C07160=1017.237,129.736,-118.733,167.035,53.865,159.921
C07161=1017.243,129.986,-118.752,167.038,53.856,159.920
C07162=1017.248,130.235,-118.770,167.040,53.847,159.919
C07163=1017.252,130.484,-118.790,167.043,53.838,159.918
C07164=1017.258,130.733,-118.809,167.046,53.829,159.917
C07165=1017.262,130.983,-118.828,167.049,53.820,159.915
C07166=1017.267,131.232,-118.847,167.052,53.811,159.914
C07167=1017.272,131.480,-118.866,167.055,53.802,159.913
C07168=1017.276,131.731,-118.885,167.058,53.793,159.912
C07169=1017.282,131.980,-118.904,167.061,53.784,159.911
C07170=1017.286,132.229,-118.923,167.065,53.774,159.910
C07171=1017.291,132.478,-118.941,167.068,53.765,159.909
C07172=1017.296,132.728,-118.961,167.071,53.756,159.907
C07173=1017.301,132.976,-118.980,167.074,53.747,159.906
C07174=1017.306,133.225,-118.999,167.077,53.738,159.905
C07175=1017.310,133.476,-119.018,167.081,53.730,159.904
C07176=1017.315,133.724,-119.037,167.084,53.721,159.903
C07177=1017.320,133.973,-119.056,167.087,53.712,159.902
C07178=1017.325,134.222,-119.075,167.091,53.702,159.901
C07179=1017.330,134.472,-119.094,167.094,53.693,159.900
C07180=1017.335,134.721,-119.113,167.097,53.684,159.898
C07181=1017.340,134.970,-119.132,167.100,53.675,159.897
C07182=1017.345,135.220,-119.152,167.103,53.666,159.896
C07183=1017.350,135.468,-119.171,167.106,53.657,159.895
C07184=1017.354,135.718,-119.189,167.110,53.648,159.894
C07185=1017.360,135.967,-119.209,167.113,53.639,159.893
C07186=1017.364,136.216,-119.228,167.116,53.630,159.892
C07187=1017.369,136.465,-119.247,167.119,53.621,159.890
C07188=1017.375,136.715,-119.266,167.122,53.612,159.889
C07189=1017.379,136.964,-119.286,167.125,53.603,159.888
C07190=1017.385,137.213,-119.305,167.128,53.594,159.887
C07191=1017.389,137.463,-119.324,167.132,53.585,159.886
C07192=1017.394,137.712,-119.343,167.135,53.576,159.885
C07193=1017.399,137.961,-119.363,167.138,53.567,159.884
C07194=1017.403,138.210,-119.382,167.141,53.558,159.882
C07195=1017.408,138.459,-119.401,167.144,53.549,159.881
C07196=1017.414,138.741,-119.423,167.148,53.538,159.880
C07197=1017.419,139.022,-119.445,167.151,53.528,159.879
C07198=1017.424,139.304,-119.467,167.155,53.518,159.877
C07199=1017.430,139.585,-119.489,167.159,53.508,159.876
C07200=1017.434,139.834,-119.508,167.162,53.499,159.875
C07201=1017.440,140.084,-119.528,167.166,53.490,159.874
C07202=1017.444,140.333,-119.547,167.169,53.481,159.873
C07203=1017.449,140.583,-119.567,167.172,53.472,159.872
C07204=1017.454,140.831,-119.586,167.175,53.464,159.871
C07205=1017.459,141.080,-119.606,167.179,53.455,159.870
C07206=1017.464,141.329,-119.626,167.182,53.446,159.868
C07207=1017.469,141.578,-119.645,167.186,53.436,159.867
C07208=1017.474,141.828,-119.665,167.189,53.427,159.866
C07209=1017.478,142.077,-119.684,167.192,53.418,159.865
C07210=1017.484,142.326,-119.703,167.195,53.409,159.864
C07211=1017.488,142.575,-119.723,167.198,53.400,159.863
C07212=1017.493,142.825,-119.743,167.201,53.391,159.862
C07213=1017.498,143.074,-119.762,167.205,53.382,159.861
C07214=1017.503,143.323,-119.781,167.208,53.373,159.859
C07215=1017.508,143.572,-119.802,167.211,53.364,159.858
C07216=1017.512,143.821,-119.821,167.214,53.355,159.857
C07217=1017.518,144.071,-119.840,167.217,53.346,159.856
C07218=1017.522,144.320,-119.860,167.222,53.337,159.855
C07219=1017.527,144.569,-119.880,167.225,53.329,159.854
C07220=1017.532,144.818,-119.898,167.228,53.320,159.853
C07221=1017.538,145.067,-119.919,167.231,53.311,159.852
C07222=1017.542,145.316,-119.939,167.234,53.302,159.850
C07223=1017.548,145.566,-119.958,167.238,53.293,159.849
C07224=1017.552,145.815,-119.977,167.242,53.284,159.848
C07225=1017.557,146.064,-119.998,167.245,53.275,159.847
C07226=1017.562,146.313,-120.017,167.248,53.266,159.846
C07227=1017.567,146.563,-120.037,167.251,53.257,159.845
C07228=1017.571,146.812,-120.057,167.255,53.247,159.844
C07229=1017.576,147.061,-120.077,167.259,53.239,159.843
C07230=1017.581,147.310,-120.097,167.262,53.230,159.842
C07231=1017.586,147.559,-120.116,167.265,53.221,159.841
C07232=1017.592,147.808,-120.136,167.268,53.212,159.839
C07233=1017.596,148.057,-120.156,167.271,53.203,159.838
C07234=1017.601,148.307,-120.176,167.275,53.194,159.837
C07235=1017.605,148.556,-120.196,167.278,53.185,159.836
C07236=1017.610,148.805,-120.216,167.282,53.177,159.835
C07237=1017.615,149.054,-120.236,167.285,53.168,159.834
C07238=1017.620,149.304,-120.256,167.288,53.159,159.833
C07239=1017.625,149.552,-120.276,167.292,53.150,159.832
C07240=1017.630,149.802,-120.296,167.295,53.141,159.831
C07241=1017.635,150.051,-120.316,167.298,53.132,159.829
C07242=1017.639,150.300,-120.336,167.302,53.123,159.828
C07243=1017.644,150.549,-120.356,167.305,53.115,159.827
C07244=1017.649,150.798,-120.376,167.309,53.105,159.826
C07245=1017.654,151.048,-120.396,167.312,53.097,159.825
C07246=1017.658,151.296,-120.416,167.316,53.088,159.824
C07247=1017.663,151.546,-120.436,167.319,53.079,159.823
C07248=1017.669,151.795,-120.456,167.323,53.069,159.822
C07249=1017.673,152.044,-120.476,167.326,53.061,159.821
C07250=1017.678,152.293,-120.496,167.330,53.052,159.820
C07251=1017.684,152.542,-120.516,167.333,53.043,159.819
C07252=1017.689,152.791,-120.536,167.336,53.035,159.818
C07253=1017.693,153.041,-120.557,167.340,53.025,159.816
C07254=1017.697,153.290,-120.576,167.343,53.016,159.815
C07255=1017.703,153.539,-120.597,167.346,53.007,159.814
C07256=1017.708,153.788,-120.617,167.350,52.999,159.813
C07257=1017.712,154.037,-120.637,167.354,52.990,159.812
C07258=1017.718,154.286,-120.657,167.357,52.981,159.811
C07259=1017.723,154.536,-120.677,167.360,52.972,159.810
C07260=1017.728,154.817,-120.701,167.364,52.962,159.809
C07261=1017.733,155.099,-120.723,167.368,52.952,159.807
C07262=1017.739,155.380,-120.746,167.372,52.942,159.806
C07263=1017.744,155.662,-120.769,167.376,52.932,159.805
C07264=1017.749,155.910,-120.789,167.380,52.924,159.804
C07265=1017.754,156.159,-120.810,167.383,52.915,159.803
C07266=1017.759,156.408,-120.830,167.386,52.906,159.802
C07267=1017.764,156.657,-120.850,167.391,52.897,159.801
C07268=1017.769,156.906,-120.870,167.394,52.888,159.800
C07269=1017.774,157.156,-120.892,167.397,52.880,159.799
C07270=1017.778,157.405,-120.911,167.401,52.871,159.798
C07271=1017.783,157.654,-120.932,167.405,52.862,159.797
C07272=1017.788,157.903,-120.952,167.408,52.853,159.795
C07273=1017.794,158.152,-120.973,167.411,52.844,159.794
C07274=1017.798,158.401,-120.992,167.415,52.835,159.793
C07275=1017.803,158.650,-121.013,167.419,52.826,159.792
C07276=1017.808,158.900,-121.034,167.422,52.818,159.791
C07277=1017.812,159.149,-121.055,167.425,52.809,159.790
C07278=1017.817,159.398,-121.075,167.429,52.801,159.789
C07279=1017.821,159.647,-121.096,167.432,52.792,159.788
C07280=1017.827,159.896,-121.117,167.437,52.783,159.787
C07281=1017.831,160.145,-121.138,167.440,52.774,159.786
C07282=1017.835,160.394,-121.159,167.444,52.766,159.785
C07283=1017.841,160.643,-121.180,167.447,52.757,159.784
C07284=1017.845,160.892,-121.201,167.450,52.748,159.783
C07285=1017.850,161.141,-121.221,167.454,52.740,159.782
C07286=1017.854,161.390,-121.243,167.458,52.731,159.781
C07287=1017.859,161.640,-121.264,167.462,52.723,159.780
C07288=1017.864,161.889,-121.284,167.465,52.714,159.779
C07289=1017.868,162.137,-121.305,167.468,52.705,159.778
C07290=1017.873,162.387,-121.326,167.472,52.697,159.777
C07291=1017.878,162.636,-121.347,167.475,52.688,159.776
C07292=1017.882,162.885,-121.368,167.480,52.680,159.775
C07293=1017.887,163.133,-121.389,167.483,52.671,159.774
C07294=1017.892,163.383,-121.410,167.486,52.662,159.772
C07295=1017.897,163.632,-121.431,167.490,52.654,159.772
C07296=1017.902,163.881,-121.452,167.494,52.645,159.771
C07297=1017.906,164.131,-121.473,167.498,52.637,159.770
C07298=1017.911,164.379,-121.493,167.501,52.628,159.768
C07299=1017.916,164.628,-121.515,167.504,52.619,159.767
C07300=1017.921,164.877,-121.535,167.508,52.611,159.766
C07301=1017.925,165.127,-121.557,167.512,52.602,159.765
C07302=1017.930,165.376,-121.578,167.516,52.593,159.764
C07303=1017.935,165.625,-121.598,167.519,52.585,159.763
C07304=1017.939,165.873,-121.620,167.523,52.575,159.762
C07305=1017.945,166.122,-121.640,167.527,52.567,159.761
C07306=1017.949,166.372,-121.662,167.530,52.558,159.760
C07307=1017.954,166.621,-121.683,167.534,52.550,159.759
C07308=1017.959,166.870,-121.704,167.538,52.541,159.758
C07309=1017.964,167.119,-121.725,167.542,52.532,159.757
C07310=1017.969,167.368,-121.746,167.545,52.524,159.756
C07311=1017.974,167.618,-121.767,167.548,52.515,159.755
C07312=1017.978,167.866,-121.788,167.553,52.506,159.754
C07313=1017.983,168.115,-121.809,167.556,52.498,159.753
C07314=1017.988,168.364,-121.830,167.560,52.489,159.752
C07315=1017.993,168.613,-121.851,167.564,52.480,159.751
C07316=1017.998,168.862,-121.872,167.568,52.472,159.750
C07317=1018.002,169.112,-121.894,167.571,52.463,159.749
C07318=1018.008,169.360,-121.915,167.575,52.454,159.748
C07319=1018.012,169.610,-121.936,167.579,52.446,159.747
C07320=1018.017,169.859,-121.957,167.582,52.437,159.746
C07321=1018.022,170.108,-121.978,167.587,52.429,159.745
C07322=1018.027,170.357,-122.000,167.590,52.420,159.744
C07323=1018.032,170.606,-122.020,167.594,52.411,159.743
C07324=1018.038,170.887,-122.044,167.598,52.401,159.742
C07325=1018.043,171.168,-122.068,167.603,52.392,159.741
C07326=1018.048,171.449,-122.092,167.607,52.382,159.739
C07327=1018.054,171.731,-122.116,167.611,52.372,159.738
C07328=1018.058,171.980,-122.137,167.615,52.364,159.737
C07329=1018.064,172.228,-122.158,167.618,52.355,159.736
C07330=1018.069,172.478,-122.180,167.623,52.346,159.735
C07331=1018.074,172.727,-122.201,167.627,52.338,159.734
C07332=1018.079,172.976,-122.222,167.630,52.329,159.733
C07333=1018.084,173.225,-122.244,167.634,52.320,159.732
C07334=1018.089,173.474,-122.265,167.638,52.312,159.731
C07335=1018.094,173.723,-122.287,167.642,52.302,159.730
C07336=1018.098,173.972,-122.308,167.645,52.294,159.729
C07337=1018.104,174.221,-122.329,167.649,52.286,159.728
C07338=1018.108,174.470,-122.350,167.654,52.276,159.727
C07339=1018.114,174.719,-122.371,167.657,52.268,159.726
C07340=1018.118,174.968,-122.393,167.662,52.259,159.725
C07341=1018.123,175.217,-122.414,167.665,52.250,159.724
C07342=1018.129,175.466,-122.435,167.669,52.241,159.723
C07343=1018.133,175.715,-122.457,167.673,52.233,159.722
C07344=1018.138,175.964,-122.478,167.676,52.225,159.721
C07345=1018.143,176.213,-122.499,167.681,52.215,159.720
C07346=1018.148,176.462,-122.521,167.684,52.207,159.719
C07347=1018.154,176.711,-122.542,167.689,52.198,159.718
C07348=1018.159,176.960,-122.564,167.692,52.190,159.717
C07349=1018.163,177.210,-122.585,167.697,52.181,159.716
C07350=1018.169,177.458,-122.606,167.700,52.172,159.715
C07351=1018.174,177.707,-122.628,167.705,52.164,159.714
C07352=1018.178,177.956,-122.649,167.708,52.155,159.713
C07353=1018.184,178.205,-122.671,167.713,52.146,159.712
C07354=1018.189,178.454,-122.693,167.716,52.138,159.711
C07355=1018.194,178.704,-122.714,167.721,52.129,159.710
C07356=1018.199,178.952,-122.735,167.724,52.120,159.709
C07357=1018.204,179.201,-122.757,167.729,52.112,159.708
C07358=1018.210,179.450,-122.778,167.732,52.103,159.707
C07359=1018.214,179.699,-122.800,167.737,52.094,159.706
C07360=1018.220,179.949,-122.822,167.740,52.086,159.705
C07361=1018.225,180.198,-122.842,167.745,52.077,159.704
C07362=1018.230,180.447,-122.864,167.748,52.068,159.703
C07363=1018.235,180.695,-122.886,167.753,52.060,159.702
C07364=1018.240,180.944,-122.907,167.756,52.051,159.701
C07365=1018.245,181.194,-122.929,167.761,52.042,159.700
C07366=1018.250,181.443,-122.951,167.764,52.034,159.699
C07367=1018.256,181.691,-122.972,167.769,52.025,159.698
C07368=1018.261,181.940,-122.994,167.772,52.016,159.697
C07369=1018.266,182.190,-123.016,167.777,52.008,159.696
C07370=1018.270,182.439,-123.039,167.781,52.000,159.695
C07371=1018.275,182.688,-123.060,167.785,51.991,159.694
C07372=1018.280,182.937,-123.082,167.789,51.983,159.693
C07373=1018.284,183.186,-123.105,167.793,51.975,159.692
C07374=1018.289,183.435,-123.127,167.797,51.965,159.691
C07375=1018.294,183.684,-123.149,167.801,51.957,159.690
C07376=1018.299,183.933,-123.171,167.805,51.949,159.689
C07377=1018.303,184.182,-123.193,167.809,51.941,159.688
C07378=1018.309,184.431,-123.216,167.813,51.932,159.687
C07379=1018.314,184.680,-123.238,167.818,51.924,159.686
C07380=1018.318,184.928,-123.260,167.821,51.916,159.685
C07381=1018.322,185.178,-123.282,167.825,51.907,159.684
C07382=1018.328,185.427,-123.305,167.830,51.899,159.684
C07383=1018.333,185.675,-123.327,167.833,51.891,159.683
C07384=1018.337,185.924,-123.350,167.838,51.882,159.682
C07385=1018.342,186.173,-123.371,167.842,51.874,159.681
C07386=1018.347,186.423,-123.394,167.846,51.865,159.680
C07387=1018.351,186.672,-123.416,167.850,51.857,159.679
C07388=1018.357,186.952,-123.441,167.854,51.848,159.678
C07389=1018.363,187.233,-123.467,167.860,51.838,159.677
C07390=1018.368,187.514,-123.492,167.864,51.829,159.676
C07391=1018.374,187.794,-123.517,167.869,51.819,159.675
C07392=1018.379,188.044,-123.539,167.872,51.811,159.674
C07393=1018.384,188.292,-123.561,167.877,51.802,159.673
C07394=1018.388,188.541,-123.584,167.881,51.794,159.672
C07395=1018.394,188.790,-123.607,167.886,51.785,159.671
C07396=1018.398,189.039,-123.629,167.889,51.777,159.670
C07397=1018.403,189.288,-123.652,167.894,51.769,159.669
C07398=1018.408,189.537,-123.674,167.898,51.761,159.668
C07399=1018.413,189.786,-123.696,167.903,51.752,159.667
C07400=1018.419,190.035,-123.719,167.906,51.744,159.666
C07401=1018.423,190.284,-123.741,167.911,51.736,159.665
C07402=1018.428,190.533,-123.763,167.915,51.727,159.664
C07403=1018.433,190.782,-123.786,167.919,51.719,159.663
C07404=1018.438,191.031,-123.808,167.923,51.711,159.662
C07405=1018.443,191.280,-123.831,167.928,51.702,159.661
C07406=1018.448,191.529,-123.853,167.932,51.694,159.661
C07407=1018.453,191.777,-123.876,167.936,51.685,159.660
C07408=1018.458,192.027,-123.899,167.940,51.677,159.659
C07409=1018.463,192.275,-123.921,167.945,51.668,159.658
C07410=1018.468,192.525,-123.944,167.949,51.660,159.657
C07411=1018.473,192.773,-123.966,167.953,51.651,159.656
C07412=1018.478,193.022,-123.989,167.958,51.643,159.655
C07413=1018.483,193.271,-124.011,167.962,51.635,159.654
C07414=1018.488,193.520,-124.034,167.967,51.627,159.653
C07415=1018.493,193.769,-124.056,167.970,51.618,159.652
C07416=1018.498,194.017,-124.079,167.975,51.610,159.651
C07417=1018.503,194.267,-124.102,167.980,51.602,159.651
C07418=1018.508,194.515,-124.124,167.983,51.593,159.649
C07419=1018.514,194.764,-124.147,167.988,51.585,159.649
C07420=1018.518,195.014,-124.170,167.992,51.577,159.648
C07421=1018.523,195.262,-124.192,167.996,51.568,159.647
C07422=1018.529,195.512,-124.215,168.001,51.559,159.646
C07423=1018.533,195.760,-124.238,168.005,51.551,159.645
C07424=1018.539,196.009,-124.261,168.010,51.543,159.644
C07425=1018.544,196.258,-124.283,168.013,51.535,159.643
C07426=1018.549,196.507,-124.306,168.018,51.526,159.642
C07427=1018.554,196.756,-124.328,168.023,51.518,159.641
C07428=1018.559,197.005,-124.351,168.027,51.509,159.640
C07429=1018.564,197.253,-124.374,168.032,51.501,159.639
C07430=1018.569,197.503,-124.396,168.036,51.493,159.639
C07431=1018.575,197.752,-124.419,168.040,51.485,159.638
C07432=1018.580,198.000,-124.442,168.045,51.476,159.637
C07433=1018.585,198.249,-124.466,168.050,51.468,159.636
C07434=1018.590,198.498,-124.487,168.054,51.460,159.635
C07435=1018.596,198.747,-124.510,168.058,51.451,159.634
C07436=1018.601,198.996,-124.534,168.063,51.442,159.633
C07437=1018.605,199.245,-124.556,168.068,51.434,159.632
C07438=1018.610,199.494,-124.579,168.072,51.426,159.631
C07439=1018.616,199.743,-124.602,168.077,51.418,159.630
C07440=1018.621,199.992,-124.625,168.081,51.410,159.630
C07441=1018.625,200.241,-124.649,168.085,51.402,159.629
C07442=1018.631,200.490,-124.672,168.090,51.393,159.628
C07443=1018.636,200.738,-124.695,168.094,51.385,159.627
C07444=1018.641,200.987,-124.719,168.099,51.377,159.626
C07445=1018.645,201.236,-124.742,168.103,51.369,159.625
C07446=1018.651,201.485,-124.765,168.108,51.361,159.624
C07447=1018.656,201.734,-124.788,168.112,51.352,159.623
C07448=1018.660,201.983,-124.811,168.116,51.344,159.622
C07449=1018.666,202.231,-124.834,168.121,51.336,159.622
C07450=1018.671,202.481,-124.858,168.126,51.328,159.621
C07451=1018.675,202.729,-124.881,168.130,51.320,159.620
C07452=1018.702,203.979,-125.000,168.600,51.411,159.725
C07453=1018.707,204.207,-125.023,168.603,51.404,159.724
C07454=1018.713,204.434,-125.045,168.607,51.398,159.723
C07455=1018.718,204.661,-125.068,168.610,51.391,159.723
C07456=1018.724,204.888,-125.090,168.614,51.385,159.722
C07457=1018.730,205.116,-125.113,168.617,51.378,159.721
C07458=1018.735,205.343,-125.137,168.620,51.372,159.720
C07459=1018.740,205.570,-125.159,168.624,51.365,159.720
C07460=1018.747,205.819,-125.184,168.628,51.358,159.719
C07461=1018.753,206.068,-125.209,168.631,51.351,159.718
C07462=1018.758,206.316,-125.234,168.635,51.343,159.717
C07463=1018.764,206.565,-125.259,168.640,51.336,159.716
C07464=1018.771,206.813,-125.284,168.643,51.329,159.715
C07465=1018.777,207.062,-125.310,168.647,51.322,159.715
C07466=1018.782,207.311,-125.334,168.650,51.315,159.714
C07467=1018.788,207.559,-125.359,168.655,51.308,159.713
C07468=1018.794,207.808,-125.385,168.658,51.301,159.712
C07469=1018.801,208.057,-125.410,168.662,51.294,159.711
C07470=1018.806,208.305,-125.435,168.666,51.287,159.711
C07471=1018.812,208.554,-125.460,168.670,51.280,159.710
C07472=1018.818,208.803,-125.485,168.674,51.273,159.709
C07473=1018.824,209.052,-125.511,168.677,51.266,159.708
C07474=1018.830,209.300,-125.536,168.682,51.260,159.707
C07475=1018.836,209.548,-125.561,168.685,51.253,159.707
C07476=1018.842,209.797,-125.586,168.689,51.246,159.706
C07477=1018.848,210.046,-125.612,168.692,51.239,159.705
C07478=1018.854,210.294,-125.637,168.697,51.232,159.704
C07479=1018.860,210.543,-125.663,168.700,51.225,159.703
C07480=1018.866,210.792,-125.688,168.705,51.218,159.703
C07481=1018.872,211.040,-125.713,168.708,51.212,159.702
C07482=1018.878,211.289,-125.739,168.712,51.204,159.701
C07483=1018.883,211.538,-125.765,168.715,51.198,159.700
C07484=1018.889,211.786,-125.790,168.720,51.191,159.700
C07485=1018.896,212.035,-125.815,168.723,51.184,159.699
C07486=1018.901,212.284,-125.841,168.728,51.177,159.698
C07487=1018.907,212.533,-125.867,168.731,51.170,159.697
C07488=1018.913,212.781,-125.892,168.735,51.164,159.696
C07489=1018.919,213.029,-125.917,168.739,51.157,159.696
C07490=1018.925,213.278,-125.943,168.742,51.150,159.695
C07491=1018.931,213.527,-125.968,168.747,51.144,159.694
C07492=1018.937,213.775,-125.994,168.750,51.137,159.693
C07493=1018.942,214.024,-126.019,168.754,51.130,159.693
C07494=1018.949,214.273,-126.045,168.758,51.124,159.692
C07495=1018.955,214.521,-126.071,168.762,51.117,159.691
C07496=1018.961,214.770,-126.096,168.765,51.110,159.690
C07497=1018.967,215.019,-126.122,168.770,51.103,159.690
C07498=1018.973,215.268,-126.147,168.773,51.096,159.689
C07499=1018.979,215.516,-126.173,168.777,51.090,159.688
C07500=1018.984,215.764,-126.198,168.781,51.083,159.687
C07501=1018.990,216.013,-126.224,168.785,51.076,159.687
C07502=1018.997,216.261,-126.250,168.789,51.070,159.686
C07503=1019.003,216.510,-126.275,168.793,51.063,159.685
C07504=1019.009,216.759,-126.301,168.797,51.057,159.685
C07505=1019.015,217.007,-126.326,168.801,51.050,159.684
C07506=1019.021,217.256,-126.352,168.805,51.043,159.683
C07507=1019.027,217.505,-126.378,168.809,51.037,159.682
C07508=1019.033,217.753,-126.404,168.812,51.031,159.682
C07509=1019.039,218.002,-126.429,168.816,51.023,159.681
C07510=1019.046,218.250,-126.455,168.820,51.017,159.680
C07511=1019.051,218.499,-126.481,168.824,51.010,159.679
C07512=1019.057,218.726,-126.505,168.827,51.004,159.679
C07513=1019.062,218.955,-126.528,168.831,50.999,159.678
C07514=1019.068,219.183,-126.552,168.835,50.993,159.677
C07515=1019.073,219.411,-126.577,168.839,50.987,159.677
C07516=1019.078,219.639,-126.600,168.842,50.981,159.676
C07517=1019.084,219.867,-126.624,168.846,50.975,159.676
C07518=1019.089,220.095,-126.648,168.849,50.969,159.675
C07519=1019.095,220.322,-126.672,168.853,50.963,159.674
C07520=1019.100,220.571,-126.698,168.856,50.957,159.674
C07521=1019.107,220.819,-126.724,168.861,50.950,159.673
C07522=1019.112,221.068,-126.750,168.864,50.944,159.672
C07523=1019.118,221.317,-126.777,168.868,50.938,159.671
C07524=1019.124,221.565,-126.802,168.873,50.931,159.671
C07525=1019.131,221.814,-126.829,168.876,50.925,159.670
C07526=1019.137,222.063,-126.854,168.880,50.919,159.669
C07527=1019.143,222.311,-126.881,168.884,50.912,159.669
C07528=1019.148,222.560,-126.907,168.888,50.906,159.668
C07529=1019.155,222.808,-126.933,168.892,50.900,159.667
C07530=1019.160,223.057,-126.959,168.897,50.894,159.667
C07531=1019.167,223.305,-126.985,168.900,50.887,159.666
C07532=1019.172,223.554,-127.012,168.904,50.881,159.665
C07533=1019.178,223.803,-127.038,168.908,50.874,159.665
C07534=1019.185,224.052,-127.064,168.912,50.868,159.664
C07535=1019.190,224.300,-127.090,168.916,50.862,159.663
C07536=1019.197,224.549,-127.116,168.920,50.856,159.663
C07537=1019.203,224.797,-127.143,168.924,50.850,159.662
C07538=1019.208,225.046,-127.168,168.928,50.843,159.662
C07539=1019.215,225.294,-127.195,168.932,50.836,159.661
C07540=1019.220,225.542,-127.221,168.936,50.830,159.660
C07541=1019.227,225.792,-127.247,168.940,50.824,159.659
C07542=1019.233,226.040,-127.274,168.944,50.818,159.659
C07543=1019.239,226.288,-127.300,168.948,50.812,159.658
C07544=1019.245,226.536,-127.326,168.952,50.806,159.658
C07545=1019.251,226.785,-127.352,168.955,50.800,159.657
C07546=1019.257,227.034,-127.379,168.960,50.793,159.656
C07547=1019.263,227.283,-127.406,168.964,50.787,159.656
C07548=1019.269,227.531,-127.432,168.967,50.781,159.655
C07549=1019.275,227.779,-127.459,168.972,50.776,159.655
C07550=1019.281,228.028,-127.485,168.976,50.769,159.654
C07551=1019.287,228.276,-127.512,168.980,50.763,159.653
C07552=1019.293,228.526,-127.538,168.984,50.757,159.653
C07553=1019.299,228.774,-127.565,168.987,50.751,159.652
C07554=1019.305,229.022,-127.591,168.992,50.745,159.651
C07555=1019.311,229.270,-127.617,168.996,50.738,159.651
C07556=1019.317,229.519,-127.645,169.000,50.733,159.650
C07557=1019.323,229.768,-127.671,169.004,50.727,159.650
C07558=1019.329,230.016,-127.698,169.007,50.721,159.649
C07559=1019.335,230.265,-127.724,169.012,50.715,159.648
C07560=1019.341,230.514,-127.751,169.016,50.709,159.648
C07561=1019.347,230.762,-127.778,169.020,50.703,159.647
C07562=1019.353,231.010,-127.805,169.024,50.697,159.647
C07563=1019.358,231.259,-127.831,169.028,50.692,159.646
C07564=1019.365,231.508,-127.858,169.033,50.685,159.646
C07565=1019.371,231.755,-127.886,169.036,50.679,159.645
C07566=1019.377,232.004,-127.912,169.040,50.674,159.644
C07567=1019.383,232.253,-127.939,169.044,50.668,159.644
C07568=1019.389,232.501,-127.966,169.048,50.662,159.643
C07569=1019.394,232.750,-127.993,169.053,50.656,159.643
C07570=1019.400,232.998,-128.019,169.057,50.650,159.642
C07571=1019.407,233.247,-128.046,169.060,50.644,159.641
C07572=1019.412,233.470,-128.071,169.064,50.639,159.641
C07573=1019.418,233.695,-128.095,169.068,50.633,159.640
C07574=1019.423,233.918,-128.119,169.072,50.628,159.640
C07575=1019.429,234.143,-128.143,169.075,50.623,159.639
C07576=1019.434,234.366,-128.167,169.079,50.618,159.639
C07577=1019.440,234.590,-128.192,169.082,50.613,159.638
C07578=1019.445,234.814,-128.216,169.086,50.607,159.638
C07579=1019.450,235.038,-128.241,169.089,50.602,159.637
C07580=1019.456,235.286,-128.268,169.094,50.596,159.637
C07581=1019.462,235.534,-128.294,169.098,50.590,159.636
C07582=1019.468,235.783,-128.322,169.102,50.585,159.636
C07583=1019.474,236.031,-128.349,169.106,50.579,159.635
C07584=1019.481,236.280,-128.376,169.110,50.574,159.635
C07585=1019.487,236.528,-128.403,169.114,50.568,159.634
C07586=1019.492,236.776,-128.430,169.119,50.562,159.634
C07587=1019.499,237.025,-128.457,169.123,50.556,159.633
C07588=1019.505,237.273,-128.484,169.127,50.551,159.632
C07589=1019.511,237.522,-128.511,169.131,50.545,159.632
C07590=1019.517,237.771,-128.538,169.135,50.539,159.631
C07591=1019.524,238.019,-128.566,169.139,50.534,159.631
C07592=1019.529,238.267,-128.592,169.144,50.527,159.630
C07593=1019.535,238.516,-128.619,169.148,50.522,159.630
C07594=1019.541,238.765,-128.647,169.152,50.517,159.629
C07595=1019.547,239.013,-128.674,169.156,50.511,159.629
C07596=1019.554,239.261,-128.702,169.160,50.505,159.628
C07597=1019.559,239.510,-128.728,169.164,50.500,159.628
C07598=1019.565,239.758,-128.756,169.168,50.495,159.627
C07599=1019.571,240.007,-128.783,169.172,50.489,159.627
C07600=1019.578,240.255,-128.811,169.176,50.483,159.626
C07601=1019.583,240.503,-128.839,169.180,50.478,159.626
C07602=1019.590,240.752,-128.866,169.185,50.472,159.625
C07603=1019.596,241.000,-128.893,169.189,50.467,159.625
C07604=1019.602,241.249,-128.922,169.194,50.461,159.624
C07605=1019.607,241.497,-128.948,169.197,50.455,159.624
C07606=1019.614,241.746,-128.976,169.201,50.450,159.623
C07607=1019.619,241.994,-129.004,169.206,50.445,159.623
C07608=1019.626,242.243,-129.031,169.210,50.439,159.622
C07609=1019.632,242.491,-129.058,169.214,50.434,159.622
C07610=1019.638,242.739,-129.087,169.218,50.429,159.621
C07611=1019.644,242.988,-129.113,169.222,50.423,159.621
C07612=1019.650,243.236,-129.141,169.226,50.418,159.620
C07613=1019.656,243.484,-129.169,169.230,50.413,159.620
C07614=1019.661,243.733,-129.197,169.235,50.407,159.620
C07615=1019.668,243.981,-129.225,169.239,50.402,159.619
C07616=1019.673,244.230,-129.252,169.243,50.397,159.619
C07617=1019.679,244.478,-129.280,169.247,50.391,159.618
C07618=1019.685,244.726,-129.308,169.251,50.386,159.618
C07619=1019.691,244.975,-129.336,169.255,50.381,159.617
C07620=1019.697,245.223,-129.364,169.259,50.375,159.617
C07621=1019.703,245.472,-129.392,169.264,50.370,159.616
C07622=1019.709,245.720,-129.420,169.268,50.365,159.616
C07623=1019.715,245.968,-129.448,169.272,50.360,159.616
C07624=1019.721,246.217,-129.476,169.276,50.355,159.615
C07625=1019.726,246.465,-129.504,169.280,50.349,159.615
C07626=1019.733,246.713,-129.532,169.285,50.344,159.614
C07627=1019.739,246.962,-129.560,169.289,50.339,159.614
C07628=1019.744,247.210,-129.588,169.293,50.334,159.613
C07629=1019.751,247.459,-129.616,169.297,50.329,159.613
C07630=1019.756,247.707,-129.644,169.302,50.323,159.612
C07631=1019.762,247.956,-129.672,169.307,50.318,159.612
C07632=1019.768,248.176,-129.696,169.310,50.313,159.612
C07633=1019.773,248.397,-129.722,169.314,50.309,159.611
C07634=1019.779,248.617,-129.746,169.318,50.304,159.611
C07635=1019.784,248.838,-129.771,169.321,50.299,159.610
C07636=1019.790,249.059,-129.796,169.325,50.295,159.610
C07637=1019.794,249.279,-129.821,169.330,50.290,159.610
C07638=1019.801,249.500,-129.846,169.333,50.286,159.610
C07639=1019.805,249.721,-129.871,169.337,50.282,159.609
C07640=1019.812,249.968,-129.899,169.341,50.276,159.609
C07641=1019.818,250.216,-129.927,169.345,50.271,159.608
C07642=1019.824,250.465,-129.956,169.349,50.266,159.608
C07643=1019.830,250.714,-129.983,169.354,50.261,159.607
C07644=1019.836,250.962,-130.012,169.358,50.256,159.607
C07645=1019.842,251.210,-130.040,169.362,50.251,159.607
C07646=1019.849,251.458,-130.068,169.366,50.246,159.606
C07647=1019.854,251.707,-130.096,169.371,50.240,159.606
C07648=1019.860,251.956,-130.125,169.375,50.236,159.606
C07649=1019.867,252.204,-130.152,169.379,50.230,159.605
C07650=1019.873,252.452,-130.181,169.384,50.226,159.605
C07651=1019.879,252.700,-130.210,169.388,50.220,159.604
C07652=1019.885,252.949,-130.237,169.392,50.215,159.604
C07653=1019.891,253.198,-130.266,169.397,50.210,159.604
C07654=1019.897,253.445,-130.294,169.401,50.205,159.603
C07655=1019.904,253.694,-130.322,169.405,50.200,159.603
C07656=1019.910,253.942,-130.350,169.410,50.195,159.602
C07657=1019.916,254.190,-130.379,169.414,50.191,159.602
C07658=1019.923,254.439,-130.407,169.418,50.185,159.602
C07659=1019.928,254.688,-130.435,169.423,50.181,159.601
C07660=1019.934,254.935,-130.464,169.427,50.175,159.601
C07661=1019.941,255.183,-130.492,169.431,50.171,159.601
C07662=1019.947,255.432,-130.520,169.436,50.165,159.600
C07663=1019.953,255.680,-130.549,169.440,50.161,159.600
C07664=1019.960,255.929,-130.577,169.444,50.155,159.599
C07665=1019.966,256.177,-130.606,169.449,50.151,159.599
C07666=1019.972,256.426,-130.634,169.453,50.145,159.599
C07667=1019.979,256.673,-130.663,169.458,50.141,159.598
C07668=1019.985,256.922,-130.691,169.462,50.136,159.598
C07669=1019.990,257.170,-130.719,169.467,50.131,159.598
C07670=1019.997,257.418,-130.747,169.472,50.126,159.597
C07671=1020.003,257.667,-130.776,169.476,50.121,159.597
C07672=1020.009,257.915,-130.805,169.481,50.116,159.597
C07673=1020.016,258.163,-130.833,169.485,50.111,159.596
C07674=1020.022,258.412,-130.862,169.489,50.106,159.596
C07675=1020.029,258.660,-130.891,169.494,50.101,159.596
C07676=1020.035,258.908,-130.918,169.498,50.097,159.595
C07677=1020.041,259.156,-130.947,169.503,50.091,159.595
C07678=1020.047,259.405,-130.976,169.507,50.087,159.595
C07679=1020.054,259.653,-131.004,169.512,50.082,159.594
C07680=1020.060,259.902,-131.032,169.516,50.077,159.594
C07681=1020.067,260.150,-131.062,169.520,50.072,159.594
C07682=1020.073,260.398,-131.091,169.525,50.068,159.593
C07683=1020.079,260.646,-131.120,169.529,50.063,159.593
C07684=1020.085,260.894,-131.149,169.533,50.059,159.593
C07685=1020.091,261.143,-131.177,169.538,50.054,159.592
C07686=1020.097,261.391,-131.206,169.542,50.049,159.592
C07687=1020.104,261.639,-131.235,169.547,50.045,159.592
C07688=1020.110,261.887,-131.264,169.551,50.040,159.592
C07689=1020.116,262.135,-131.293,169.556,50.036,159.591
C07690=1020.122,262.384,-131.323,169.560,50.031,159.591
C07691=1020.128,262.632,-131.352,169.565,50.026,159.591
C07692=1020.134,262.852,-131.377,169.568,50.022,159.590
C07693=1020.139,263.071,-131.403,169.572,50.018,159.590
C07694=1020.144,263.291,-131.428,169.577,50.014,159.590
C07695=1020.150,263.512,-131.454,169.580,50.010,159.590
C07696=1020.156,263.731,-131.480,169.584,50.006,159.589
C07697=1020.161,263.951,-131.506,169.588,50.002,159.589
C07698=1020.167,264.170,-131.531,169.593,49.998,159.589
C07699=1020.172,264.390,-131.557,169.596,49.993,159.589
C07700=1020.178,264.638,-131.586,169.601,49.989,159.589
C07701=1020.184,264.887,-131.615,169.606,49.985,159.588
C07702=1020.190,265.135,-131.644,169.610,49.980,159.588
C07703=1020.197,265.384,-131.674,169.615,49.976,159.588
C07704=1020.204,265.631,-131.703,169.620,49.971,159.587
C07705=1020.209,265.880,-131.733,169.624,49.966,159.587
C07706=1020.216,266.128,-131.762,169.628,49.962,159.587
C07707=1020.222,266.376,-131.791,169.633,49.958,159.587
C07708=1020.228,266.624,-131.820,169.637,49.953,159.586
C07709=1020.234,266.872,-131.850,169.642,49.949,159.586
C07710=1020.240,267.120,-131.880,169.646,49.944,159.586
C07711=1020.247,267.369,-131.909,169.651,49.940,159.586
C07712=1020.253,267.617,-131.938,169.656,49.936,159.585
C07713=1020.259,267.865,-131.968,169.660,49.931,159.585
C07714=1020.265,268.113,-131.997,169.665,49.926,159.585
C07715=1020.272,268.361,-132.026,169.670,49.923,159.585
C07716=1020.277,268.609,-132.056,169.674,49.918,159.585
C07717=1020.284,268.858,-132.085,169.678,49.914,159.584
C07718=1020.291,269.106,-132.115,169.683,49.910,159.584
C07719=1020.297,269.354,-132.144,169.687,49.905,159.584
C07720=1020.302,269.602,-132.174,169.692,49.901,159.584
C07721=1020.309,269.850,-132.204,169.697,49.897,159.583
C07722=1020.315,270.099,-132.234,169.701,49.892,159.583
C07723=1020.322,270.346,-132.263,169.706,49.888,159.583
C07724=1020.328,270.595,-132.292,169.711,49.883,159.583
C07725=1020.333,270.843,-132.322,169.716,49.879,159.583
C07726=1020.340,271.091,-132.352,169.719,49.875,159.582
C07727=1020.346,271.340,-132.382,169.724,49.871,159.582
C07728=1020.353,271.587,-132.412,169.729,49.867,159.582
C07729=1020.358,271.836,-132.441,169.733,49.862,159.582
C07730=1020.365,272.084,-132.471,169.738,49.858,159.582
C07731=1020.371,272.332,-132.500,169.743,49.854,159.581
C07732=1020.377,272.580,-132.531,169.748,49.850,159.581
C07733=1020.384,272.828,-132.561,169.753,49.846,159.581
C07734=1020.390,273.076,-132.591,169.757,49.841,159.581
C07735=1020.396,273.324,-132.620,169.761,49.837,159.581
C07736=1020.402,273.572,-132.650,169.766,49.833,159.580
C07737=1020.409,273.821,-132.680,169.771,49.829,159.580
C07738=1020.415,274.068,-132.710,169.776,49.825,159.580
C07739=1020.421,274.317,-132.739,169.780,49.820,159.580
C07740=1020.428,274.565,-132.770,169.785,49.816,159.580
C07741=1020.434,274.813,-132.800,169.790,49.813,159.580
C07742=1020.440,275.060,-132.830,169.795,49.808,159.580
C07743=1020.446,275.310,-132.860,169.800,49.804,159.579
C07744=1020.453,275.557,-132.890,169.804,49.800,159.579
C07745=1020.459,275.806,-132.921,169.808,49.796,159.579
C07746=1020.466,276.053,-132.950,169.813,49.792,159.579
C07747=1020.471,276.302,-132.980,169.818,49.788,159.579
C07748=1020.478,276.550,-133.010,169.823,49.784,159.579
C07749=1020.484,276.798,-133.041,169.828,49.779,159.578
C07750=1020.491,277.046,-133.071,169.833,49.776,159.578
C07751=1020.497,277.294,-133.101,169.838,49.772,159.578
C07752=1020.503,277.515,-133.128,169.841,49.768,159.578
C07753=1020.508,277.739,-133.155,169.845,49.764,159.578
C07754=1020.513,277.960,-133.183,169.850,49.761,159.578
C07755=1020.519,278.182,-133.210,169.855,49.758,159.578
C07756=1020.525,278.404,-133.237,169.859,49.754,159.578
C07757=1020.530,278.626,-133.264,169.862,49.750,159.577
C07758=1020.536,278.849,-133.291,169.867,49.747,159.578
C07759=1020.541,279.071,-133.319,169.872,49.743,159.577
C07760=1020.548,279.319,-133.349,169.876,49.740,159.577
C07761=1020.554,279.567,-133.379,169.881,49.736,159.577
C07762=1020.560,279.815,-133.409,169.886,49.732,159.577
C07763=1020.567,280.063,-133.441,169.890,49.728,159.577
C07764=1020.572,280.310,-133.471,169.895,49.724,159.577
C07765=1020.580,280.559,-133.501,169.900,49.720,159.577
C07766=1020.585,280.806,-133.532,169.905,49.716,159.577
C07767=1020.592,281.055,-133.562,169.910,49.712,159.577
C07768=1020.598,281.303,-133.593,169.914,49.709,159.576
C07769=1020.605,281.551,-133.623,169.919,49.705,159.576
C07770=1020.611,281.799,-133.654,169.924,49.701,159.576
C07771=1020.617,282.047,-133.685,169.929,49.697,159.576
C07772=1020.624,282.295,-133.715,169.934,49.693,159.576
C07773=1020.630,282.543,-133.746,169.939,49.689,159.576
C07774=1020.637,282.791,-133.776,169.944,49.685,159.576
C07775=1020.643,283.039,-133.807,169.949,49.682,159.576
C07776=1020.649,283.287,-133.838,169.953,49.679,159.576
C07777=1020.656,283.535,-133.868,169.958,49.675,159.576
C07778=1020.661,283.783,-133.899,169.963,49.671,159.576
C07779=1020.669,284.031,-133.929,169.968,49.667,159.576
C07780=1020.675,284.279,-133.960,169.973,49.663,159.575
C07781=1020.681,284.527,-133.991,169.978,49.660,159.576
C07782=1020.688,284.775,-134.022,169.983,49.656,159.575
C07783=1020.694,285.023,-134.052,169.988,49.652,159.575
C07784=1020.701,285.271,-134.083,169.993,49.648,159.575
C07785=1020.708,285.519,-134.114,169.997,49.645,159.575
C07786=1020.714,285.766,-134.145,170.002,49.641,159.575
C07787=1020.720,286.015,-134.176,170.007,49.637,159.575
C07788=1020.726,286.263,-134.208,170.013,49.634,159.575
C07789=1020.732,286.511,-134.238,170.017,49.630,159.575
C07790=1020.739,286.759,-134.269,170.022,49.626,159.575
C07791=1020.745,287.007,-134.300,170.028,49.623,159.575
C07792=1020.751,287.254,-134.331,170.032,49.619,159.575
C07793=1020.758,287.503,-134.362,170.037,49.616,159.575
C07794=1020.764,287.751,-134.393,170.042,49.612,159.575
C07795=1020.771,287.999,-134.425,170.047,49.608,159.575
C07796=1020.777,288.247,-134.455,170.052,49.605,159.575
C07797=1020.784,288.494,-134.487,170.057,49.601,159.575
C07798=1020.790,288.742,-134.518,170.062,49.598,159.575
C07799=1020.797,288.990,-134.550,170.067,49.594,159.575
C07800=1020.803,289.238,-134.580,170.072,49.591,159.575
C07801=1020.810,289.486,-134.611,170.077,49.588,159.575
C07802=1020.816,289.734,-134.643,170.082,49.584,159.575
C07803=1020.823,289.982,-134.674,170.087,49.581,159.575
C07804=1020.828,290.230,-134.705,170.092,49.577,159.575
C07805=1020.835,290.478,-134.737,170.098,49.573,159.575
C07806=1020.842,290.726,-134.768,170.102,49.569,159.575
C07807=1020.848,290.974,-134.799,170.108,49.566,159.575
C07808=1020.855,291.222,-134.831,170.112,49.563,159.575
C07809=1020.861,291.470,-134.862,170.117,49.559,159.575
C07810=1020.868,291.717,-134.893,170.122,49.556,159.575
C07811=1020.874,291.966,-134.925,170.128,49.553,159.575
C07812=1020.881,292.193,-134.954,170.132,49.550,159.575
C07813=1020.886,292.421,-134.982,170.137,49.546,159.575
C07814=1020.892,292.650,-135.011,170.141,49.543,159.575
C07815=1020.898,292.878,-135.041,170.147,49.540,159.575
C07816=1020.904,293.106,-135.069,170.151,49.537,159.575
C07817=1020.910,293.334,-135.099,170.155,49.534,159.575
C07818=1020.916,293.563,-135.128,170.160,49.531,159.575
C07819=1020.922,293.790,-135.157,170.165,49.528,159.575
C07820=1020.928,294.039,-135.189,170.170,49.525,159.575
C07821=1020.934,294.287,-135.221,170.175,49.521,159.576
C07822=1020.940,294.535,-135.253,170.181,49.518,159.576
C07823=1020.947,294.782,-135.285,170.186,49.515,159.576
C07824=1020.953,295.030,-135.317,170.190,49.512,159.576
C07825=1020.959,295.279,-135.349,170.196,49.509,159.576
C07826=1020.965,295.526,-135.380,170.201,49.506,159.576
C07827=1020.972,295.773,-135.413,170.206,49.502,159.576
C07828=1020.978,296.022,-135.445,170.212,49.499,159.576
C07829=1020.985,296.269,-135.476,170.217,49.496,159.576
C07830=1020.991,296.517,-135.509,170.221,49.493,159.576
C07831=1020.998,296.765,-135.540,170.227,49.490,159.576
C07832=1021.004,297.013,-135.573,170.232,49.486,159.576
C07833=1021.010,297.261,-135.605,170.237,49.483,159.577
C07834=1021.017,297.509,-135.637,170.242,49.480,159.577
C07835=1021.023,297.756,-135.669,170.248,49.477,159.577
C07836=1021.030,298.004,-135.701,170.252,49.474,159.577
C07837=1021.036,298.252,-135.733,170.258,49.471,159.577
C07838=1021.043,298.500,-135.765,170.263,49.468,159.577
C07839=1021.049,298.747,-135.798,170.268,49.465,159.577
C07840=1021.055,298.995,-135.830,170.274,49.462,159.577
C07841=1021.062,299.243,-135.862,170.279,49.458,159.577
C07842=1021.068,299.491,-135.894,170.284,49.455,159.578
C07843=1021.075,299.738,-135.926,170.290,49.452,159.578
C07844=1021.081,299.986,-135.958,170.294,49.450,159.578
C07845=1021.088,300.235,-135.991,170.300,49.446,159.578
C07846=1021.095,300.482,-136.023,170.305,49.443,159.578
C07847=1021.101,300.730,-136.055,170.311,49.441,159.578
C07848=1021.108,300.978,-136.087,170.316,49.437,159.578
C07849=1021.114,301.226,-136.119,170.321,49.434,159.579
C07850=1021.120,301.473,-136.152,170.327,49.431,159.579
C07851=1021.127,301.721,-136.184,170.332,49.428,159.579
C07852=1021.133,301.969,-136.216,170.338,49.425,159.579
C07853=1021.141,302.217,-136.249,170.342,49.422,159.579
C07854=1021.147,302.464,-136.282,170.348,49.420,159.579
C07855=1021.153,302.712,-136.314,170.353,49.416,159.579
C07856=1021.160,302.960,-136.346,170.358,49.413,159.580
C07857=1021.166,303.207,-136.379,170.364,49.410,159.580
C07858=1021.174,303.455,-136.411,170.369,49.407,159.580
C07859=1021.180,303.703,-136.444,170.374,49.404,159.580
C07860=1021.187,303.951,-136.477,170.380,49.401,159.580
C07861=1021.193,304.199,-136.508,170.385,49.398,159.580
C07862=1021.200,304.447,-136.541,170.391,49.396,159.581
C07863=1021.207,304.694,-136.573,170.396,49.392,159.581
C07864=1021.214,304.942,-136.606,170.402,49.390,159.581
C07865=1021.220,305.189,-136.639,170.407,49.387,159.581
C07866=1021.227,305.437,-136.671,170.412,49.384,159.581
C07867=1021.234,305.685,-136.704,170.417,49.381,159.581
C07868=1021.241,305.932,-136.736,170.423,49.379,159.582
C07869=1021.248,306.180,-136.769,170.428,49.375,159.582
C07870=1021.254,306.428,-136.802,170.434,49.373,159.582
C07871=1021.261,306.675,-136.834,170.439,49.370,159.582
C07872=1021.267,306.913,-136.865,170.445,49.367,159.582
C07873=1021.274,307.149,-136.896,170.450,49.364,159.583
C07874=1021.280,307.386,-136.928,170.455,49.361,159.583
C07875=1021.286,307.624,-136.959,170.461,49.359,159.583
C07876=1021.294,307.861,-136.990,170.466,49.356,159.583
C07877=1021.300,308.098,-137.022,170.471,49.353,159.583
C07878=1021.307,308.335,-137.053,170.476,49.351,159.584
C07879=1021.313,308.572,-137.084,170.482,49.348,159.584
C07880=1021.320,308.820,-137.117,170.487,49.345,159.584
C07881=1021.327,309.068,-137.150,170.493,49.342,159.584
C07882=1021.334,309.314,-137.183,170.499,49.340,159.585
C07883=1021.341,309.563,-137.216,170.504,49.337,159.585
C07884=1021.348,309.810,-137.248,170.510,49.334,159.585
C07885=1021.354,310.058,-137.281,170.515,49.331,159.585
C07886=1021.361,310.305,-137.315,170.521,49.329,159.586
C07887=1021.368,310.553,-137.348,170.527,49.326,159.586
C07888=1021.375,310.801,-137.381,170.532,49.324,159.586
C07889=1021.381,311.048,-137.414,170.537,49.322,159.586
C07890=1021.387,311.296,-137.449,170.543,49.319,159.587
C07891=1021.394,311.544,-137.481,170.548,49.316,159.587
C07892=1021.400,311.791,-137.515,170.554,49.314,159.587
C07893=1021.408,312.038,-137.549,170.560,49.311,159.587
C07894=1021.413,312.286,-137.582,170.565,49.309,159.588
C07895=1021.420,312.534,-137.616,170.571,49.306,159.588
C07896=1021.427,312.781,-137.649,170.577,49.303,159.588
C07897=1021.434,313.029,-137.682,170.583,49.301,159.589
C07898=1021.440,313.277,-137.716,170.588,49.298,159.589
C07899=1021.447,313.524,-137.750,170.594,49.296,159.589
C07900=1021.453,313.772,-137.783,170.599,49.294,159.589
C07901=1021.460,314.019,-137.817,170.605,49.292,159.590
C07902=1021.467,314.267,-137.851,170.610,49.289,159.590
C07903=1021.473,314.514,-137.885,170.616,49.286,159.590
C07904=1021.480,314.763,-137.918,170.622,49.284,159.591
C07905=1021.487,315.010,-137.951,170.627,49.281,159.591
C07906=1021.493,315.258,-137.986,170.633,49.279,159.591
C07907=1021.501,315.505,-138.019,170.639,49.277,159.592
C07908=1021.507,315.752,-138.053,170.645,49.274,159.592
C07909=1021.514,316.000,-138.087,170.650,49.272,159.592
C07910=1021.521,316.249,-138.120,170.656,49.270,159.593
C07911=1021.527,316.496,-138.154,170.662,49.267,159.593
C07912=1021.534,316.743,-138.188,170.668,49.265,159.593
C07913=1021.541,316.991,-138.222,170.674,49.263,159.594
C07914=1021.547,317.238,-138.256,170.679,49.260,159.594
C07915=1021.555,317.486,-138.289,170.685,49.257,159.594
C07916=1021.562,317.734,-138.323,170.691,49.256,159.595
C07917=1021.568,317.981,-138.357,170.697,49.253,159.595
C07918=1021.575,318.228,-138.391,170.702,49.250,159.595
C07919=1021.582,318.476,-138.425,170.709,49.248,159.596
C07920=1021.589,318.724,-138.459,170.714,49.246,159.596
C07921=1021.596,318.972,-138.493,170.720,49.244,159.597
C07922=1021.602,319.219,-138.527,170.726,49.241,159.597
C07923=1021.610,319.466,-138.560,170.732,49.239,159.597
C07924=1021.616,319.714,-138.596,170.738,49.237,159.598
C07925=1021.624,319.962,-138.629,170.743,49.234,159.598
C07926=1021.631,320.209,-138.663,170.749,49.232,159.598
C07927=1021.637,320.457,-138.698,170.755,49.230,159.599
C07928=1021.644,320.704,-138.731,170.761,49.228,159.599
C07929=1021.651,320.952,-138.765,170.767,49.226,159.600
C07930=1021.658,321.199,-138.800,170.773,49.223,159.600
C07931=1021.665,321.447,-138.834,170.779,49.221,159.600
C07932=1021.672,321.687,-138.867,170.784,49.219,159.601
C07933=1021.679,321.926,-138.900,170.790,49.217,159.601
C07934=1021.686,322.165,-138.932,170.797,49.215,159.602
C07935=1021.692,322.405,-138.966,170.802,49.212,159.602
C07936=1021.699,322.645,-138.999,170.807,49.211,159.602
C07937=1021.706,322.884,-139.032,170.813,49.209,159.603
C07938=1021.713,323.124,-139.065,170.819,49.206,159.603
C07939=1021.720,323.363,-139.099,170.825,49.204,159.604
C07940=1021.727,323.611,-139.133,170.831,49.203,159.604
C07941=1021.734,323.859,-139.167,170.837,49.200,159.604
C07942=1021.741,324.106,-139.202,170.843,49.198,159.605
C07943=1021.748,324.354,-139.235,170.849,49.196,159.605
C07944=1021.756,324.601,-139.270,170.856,49.194,159.606
C07945=1021.762,324.849,-139.304,170.861,49.191,159.606
C07946=1021.770,325.096,-139.339,170.867,49.189,159.607
C07947=1021.777,325.343,-139.373,170.873,49.187,159.607
C07948=1021.784,325.591,-139.408,170.879,49.186,159.607
C07949=1021.792,325.839,-139.442,170.886,49.184,159.608
C07950=1021.799,326.086,-139.477,170.891,49.181,159.608
C07951=1021.806,326.333,-139.512,170.897,49.179,159.609
C07952=1021.813,326.581,-139.546,170.904,49.177,159.609
C07953=1021.821,326.828,-139.580,170.910,49.175,159.610
C07954=1021.827,327.076,-139.615,170.916,49.173,159.610
C07955=1021.834,327.323,-139.650,170.922,49.171,159.611
C07956=1021.841,327.571,-139.684,170.928,49.169,159.611
C07957=1021.849,327.819,-139.720,170.934,49.167,159.612
C07958=1021.855,328.066,-139.755,170.941,49.166,159.612
C07959=1021.862,328.313,-139.790,170.947,49.164,159.613
C07960=1021.870,328.560,-139.825,170.953,49.162,159.613
C07961=1021.876,328.808,-139.860,170.959,49.160,159.614
C07962=1021.883,329.055,-139.895,170.965,49.158,159.614
C07963=1021.891,329.303,-139.930,170.972,49.156,159.615
C07964=1021.898,329.550,-139.965,170.978,49.155,159.615
C07965=1021.905,329.798,-140.000,170.984,49.153,159.616
C07966=1021.912,330.045,-140.035,170.990,49.151,159.616
C07967=1021.919,330.293,-140.071,170.996,49.149,159.617
C07968=1021.926,330.540,-140.105,171.003,49.148,159.617
C07969=1021.933,330.787,-140.140,171.009,49.146,159.618
C07970=1021.940,331.035,-140.175,171.015,49.144,159.618
C07971=1021.948,331.282,-140.212,171.022,49.141,159.619
C07972=1021.955,331.529,-140.246,171.028,49.140,159.620
C07973=1021.962,331.777,-140.281,171.034,49.138,159.620
C07974=1021.969,332.025,-140.317,171.040,49.136,159.621
C07975=1021.976,332.272,-140.352,171.047,49.135,159.621
C07976=1021.984,332.520,-140.388,171.053,49.133,159.622
C07977=1021.991,332.767,-140.423,171.059,49.132,159.622
C07978=1021.998,333.014,-140.458,171.066,49.130,159.623
C07979=1022.005,333.262,-140.493,171.073,49.128,159.624
C07980=1022.013,333.509,-140.529,171.079,49.126,159.624
C07981=1022.019,333.756,-140.564,171.085,49.125,159.625
C07982=1022.027,334.004,-140.601,171.091,49.123,159.625
C07983=1022.034,334.251,-140.636,171.097,49.122,159.626
C07984=1022.041,334.498,-140.672,171.104,49.120,159.626
C07985=1022.048,334.746,-140.707,171.111,49.118,159.627
C07986=1022.056,334.993,-140.743,171.117,49.117,159.628
C07987=1022.063,335.241,-140.778,171.123,49.115,159.628
C07988=1022.070,335.487,-140.814,171.130,49.114,159.629
C07989=1022.077,335.735,-140.850,171.136,49.112,159.629
C07990=1022.084,335.982,-140.886,171.143,49.110,159.630
C07991=1022.092,336.230,-140.922,171.149,49.109,159.631
C07992=1022.099,336.467,-140.956,171.156,49.108,159.631
C07993=1022.105,336.705,-140.990,171.162,49.106,159.632
C07994=1022.112,336.942,-141.025,171.168,49.104,159.632
C07995=1022.120,337.179,-141.059,171.175,49.103,159.633
C07996=1022.127,337.417,-141.094,171.181,49.102,159.634
C07997=1022.134,337.653,-141.128,171.187,49.100,159.634
C07998=1022.140,337.891,-141.163,171.193,49.099,159.635
C07999=1022.148,338.128,-141.197,171.200,49.097,159.636
C08000=1022.155,338.375,-141.233,171.206,49.096,159.636
C08001=1022.162,338.623,-141.269,171.213,49.095,159.637
C08002=1022.170,338.871,-141.305,171.219,49.093,159.638
C08003=1022.177,339.117,-141.341,171.226,49.091,159.638
C08004=1022.185,339.365,-141.377,171.232,49.090,159.639
C08005=1022.192,339.612,-141.413,171.239,49.088,159.639
C08006=1022.199,339.859,-141.449,171.245,49.087,159.640
C08007=1022.206,340.107,-141.486,171.252,49.086,159.641
C08008=1022.214,340.354,-141.522,171.259,49.084,159.642
C08009=1022.221,340.601,-141.558,171.266,49.084,159.642
C08010=1022.229,340.848,-141.594,171.272,49.082,159.643
C08011=1022.236,341.096,-141.631,171.279,49.081,159.644
C08012=1022.244,341.343,-141.668,171.286,49.079,159.644
C08013=1022.251,341.590,-141.704,171.292,49.078,159.645
C08014=1022.258,341.837,-141.740,171.299,49.077,159.646
C08015=1022.265,342.085,-141.777,171.306,49.075,159.647
C08016=1022.273,342.332,-141.813,171.313,49.074,159.647
C08017=1022.280,342.578,-141.850,171.319,49.073,159.648
C08018=1022.287,342.826,-141.886,171.326,49.072,159.649
C08019=1022.295,343.074,-141.923,171.333,49.070,159.649
C08020=1022.303,343.320,-141.960,171.340,49.070,159.650
C08021=1022.310,343.568,-141.996,171.347,49.068,159.651
C08022=1022.317,343.815,-142.032,171.353,49.067,159.652
C08023=1022.325,344.062,-142.069,171.360,49.066,159.653
C08024=1022.332,344.310,-142.106,171.367,49.064,159.653
C08025=1022.340,344.556,-142.143,171.374,49.063,159.654
C08026=1022.348,344.804,-142.179,171.381,49.062,159.655
C08027=1022.355,345.051,-142.217,171.388,49.061,159.656
C08028=1022.363,345.298,-142.253,171.395,49.060,159.656
C08029=1022.370,345.545,-142.290,171.401,49.059,159.657
C08030=1022.378,345.793,-142.327,171.408,49.057,159.658
C08031=1022.385,346.040,-142.364,171.415,49.056,159.659
C08032=1022.393,346.287,-142.401,171.422,49.055,159.659
C08033=1022.400,346.534,-142.437,171.429,49.054,159.660
C08034=1022.408,346.781,-142.474,171.436,49.053,159.661
C08035=1022.416,347.028,-142.512,171.443,49.052,159.662
C08036=1022.423,347.276,-142.548,171.450,49.051,159.663
C08037=1022.431,347.523,-142.586,171.456,49.050,159.663
C08038=1022.439,347.770,-142.622,171.464,49.049,159.664
C08039=1022.446,348.017,-142.660,171.471,49.048,159.665
C08040=1022.454,348.264,-142.697,171.477,49.047,159.666
C08041=1022.461,348.511,-142.734,171.485,49.046,159.667
C08042=1022.469,348.758,-142.771,171.492,49.045,159.668
C08043=1022.476,349.005,-142.808,171.500,49.044,159.669
C08044=1022.483,349.253,-142.846,171.506,49.043,159.669
C08045=1022.491,349.499,-142.883,171.514,49.042,159.670
C08046=1022.498,349.746,-142.920,171.520,49.041,159.671
C08047=1022.506,349.994,-142.958,171.527,49.040,159.672
C08048=1022.514,350.241,-142.995,171.535,49.039,159.673
C08049=1022.521,350.488,-143.033,171.542,49.039,159.674
C08050=1022.529,350.735,-143.071,171.549,49.038,159.675
C08051=1022.537,350.982,-143.108,171.556,49.036,159.675
C08052=1022.545,351.218,-143.144,171.562,49.036,159.676
C08053=1022.552,351.453,-143.180,171.569,49.035,159.677
C08054=1022.559,351.689,-143.215,171.577,49.034,159.678
C08055=1022.567,351.926,-143.250,171.584,49.033,159.679
C08056=1022.573,352.161,-143.287,171.590,49.033,159.680
C08057=1022.581,352.396,-143.323,171.597,49.032,159.681
C08058=1022.589,352.632,-143.359,171.604,49.031,159.681
C08059=1022.596,352.868,-143.395,171.612,49.030,159.682
C08060=1022.604,353.115,-143.432,171.618,49.030,159.683
C08061=1022.612,353.362,-143.470,171.626,49.029,159.684
C08062=1022.619,353.609,-143.508,171.633,49.028,159.685
C08063=1022.628,353.857,-143.545,171.641,49.027,159.686
C08064=1022.635,354.103,-143.584,171.647,49.026,159.687
C08065=1022.642,354.350,-143.621,171.655,49.026,159.688
C08066=1022.651,354.597,-143.659,171.662,49.025,159.689
C08067=1022.659,354.844,-143.697,171.670,49.024,159.690
C08068=1022.666,355.091,-143.735,171.677,49.024,159.691
C08069=1022.674,355.339,-143.773,171.685,49.023,159.692
C08070=1022.682,355.585,-143.811,171.692,49.022,159.693
C08071=1022.690,355.832,-143.850,171.699,49.022,159.694
C08072=1022.698,356.079,-143.887,171.707,49.021,159.695
C08073=1022.706,356.326,-143.925,171.714,49.020,159.695
C08074=1022.713,356.573,-143.963,171.722,49.020,159.697
C08075=1022.722,356.820,-144.002,171.729,49.019,159.697
C08076=1022.729,357.067,-144.040,171.737,49.019,159.699
C08077=1022.737,357.314,-144.078,171.745,49.018,159.699
C08078=1022.744,357.561,-144.116,171.752,49.018,159.701
C08079=1022.753,357.808,-144.154,171.759,49.017,159.701
C08080=1022.761,358.054,-144.193,171.766,49.017,159.703
C08081=1022.769,358.302,-144.231,171.774,49.016,159.703
C08082=1022.777,358.548,-144.269,171.782,49.015,159.705
C08083=1022.785,358.795,-144.308,171.789,49.015,159.706
C08084=1022.793,359.042,-144.347,171.797,49.014,159.707
C08085=1022.800,359.289,-144.385,171.805,49.014,159.708
C08086=1022.809,359.536,-144.424,171.812,49.014,159.709
C08087=1022.817,359.783,-144.462,171.820,49.013,159.710
C08088=1022.824,360.030,-144.500,171.828,49.012,159.711
C08089=1022.832,360.277,-144.539,171.835,49.012,159.712
C08090=1022.840,360.524,-144.577,171.843,49.012,159.713
C08091=1022.848,360.770,-144.617,171.851,49.011,159.714
C08092=1022.857,361.017,-144.655,171.858,49.011,159.715
C08093=1022.863,361.264,-144.694,171.866,49.010,159.716
C08094=1022.872,361.511,-144.733,171.874,49.010,159.717
C08095=1022.880,361.758,-144.772,171.881,49.010,159.718
C08096=1022.888,362.005,-144.811,171.889,49.009,159.719
C08097=1022.896,362.251,-144.850,171.898,49.009,159.721
C08098=1022.904,362.498,-144.888,171.905,49.009,159.722
C08099=1022.912,362.745,-144.928,171.913,49.008,159.723
C08100=1022.920,362.993,-144.967,171.921,49.008,159.724
C08101=1022.929,363.239,-145.006,171.929,49.008,159.725
C08102=1022.936,363.486,-145.044,171.936,49.007,159.726
C08103=1022.945,363.732,-145.084,171.944,49.008,159.727
C08104=1022.953,363.979,-145.123,171.953,49.007,159.729
C08105=1022.960,364.226,-145.162,171.961,49.007,159.730
C08106=1022.969,364.473,-145.201,171.968,49.007,159.731
C08107=1022.977,364.720,-145.241,171.976,49.006,159.732
C08108=1022.985,364.967,-145.279,171.984,49.006,159.733
C08109=1022.994,365.213,-145.319,171.992,49.006,159.734
C08110=1023.002,365.460,-145.359,172.000,49.006,159.735
C08111=1023.010,365.706,-145.398,172.008,49.005,159.737
C08112=1023.018,365.946,-145.435,172.016,49.005,159.738
C08113=1023.026,366.185,-145.474,172.024,49.005,159.739
C08114=1023.034,366.425,-145.512,172.031,49.005,159.740
C08115=1023.042,366.664,-145.550,172.039,49.005,159.741
C08116=1023.050,366.903,-145.588,172.047,49.004,159.742
C08117=1023.059,367.142,-145.626,172.055,49.005,159.744
C08118=1023.066,367.381,-145.664,172.063,49.004,159.745
C08119=1023.074,367.620,-145.703,172.071,49.004,159.746
C08120=1023.083,367.867,-145.742,172.079,49.004,159.747
C08121=1023.091,368.114,-145.781,172.087,49.004,159.748
C08122=1023.099,368.360,-145.821,172.096,49.004,159.750
C08123=1023.107,368.607,-145.860,172.103,49.005,159.751
C08124=1023.116,368.854,-145.901,172.111,49.004,159.752
C08125=1023.124,369.101,-145.941,172.120,49.004,159.753
C08126=1023.132,369.348,-145.981,172.128,49.004,159.755
C08127=1023.141,369.593,-146.021,172.136,49.004,159.756
C08128=1023.149,369.840,-146.061,172.145,49.004,159.757
C08129=1023.157,370.087,-146.100,172.153,49.004,159.758
C08130=1023.165,370.333,-146.141,172.162,49.005,159.760
C08131=1023.174,370.581,-146.180,172.170,49.005,159.761
C08132=1023.182,370.827,-146.221,172.179,49.005,159.762
C08133=1023.191,371.073,-146.260,172.187,49.005,159.764
C08134=1023.199,371.320,-146.301,172.195,49.005,159.765
C08135=1023.208,371.567,-146.341,172.204,49.005,159.766
C08136=1023.216,371.813,-146.381,172.212,49.005,159.768
C08137=1023.224,372.060,-146.421,172.220,49.005,159.769
C08138=1023.233,372.307,-146.462,172.229,49.005,159.770
C08139=1023.242,372.553,-146.502,172.237,49.006,159.772
C08140=1023.249,372.800,-146.541,172.246,49.006,159.773
C08141=1023.259,373.046,-146.582,172.254,49.006,159.774
C08142=1023.267,373.293,-146.623,172.263,49.006,159.776
C08143=1023.275,373.539,-146.663,172.271,49.006,159.777
C08144=1023.284,373.786,-146.703,172.280,49.007,159.778
C08145=1023.292,374.033,-146.743,172.288,49.007,159.780
C08146=1023.301,374.279,-146.784,172.297,49.007,159.781
C08147=1023.309,374.526,-146.825,172.305,49.008,159.782
C08148=1023.319,374.772,-146.865,172.314,49.008,159.784
C08149=1023.327,375.019,-146.906,172.323,49.008,159.785
C08150=1023.336,375.265,-146.946,172.332,49.008,159.787
C08151=1023.344,375.511,-146.987,172.340,49.008,159.788
C08152=1023.353,375.758,-147.027,172.349,49.009,159.790
C08153=1023.361,376.004,-147.068,172.358,49.009,159.791
C08154=1023.371,376.251,-147.108,172.366,49.010,159.792
C08155=1023.379,376.498,-147.149,172.376,49.010,159.794
C08156=1023.387,376.744,-147.190,172.384,49.010,159.795
C08157=1023.397,376.990,-147.231,172.393,49.011,159.797
C08158=1023.405,377.237,-147.271,172.401,49.011,159.798
C08159=1023.414,377.484,-147.312,172.410,49.012,159.800
C08160=1023.423,377.730,-147.354,172.419,49.013,159.801
C08161=1023.431,377.976,-147.395,172.429,49.012,159.802
C08162=1023.440,378.223,-147.437,172.437,49.013,159.804
C08163=1023.448,378.470,-147.478,172.446,49.014,159.806
C08164=1023.457,378.715,-147.519,172.455,49.014,159.807
C08165=1023.466,378.962,-147.559,172.464,49.014,159.808
C08166=1023.475,379.208,-147.601,172.473,49.015,159.810
C08167=1023.483,379.455,-147.642,172.482,49.016,159.812
C08168=1023.492,379.701,-147.683,172.490,49.016,159.813
C08169=1023.501,379.947,-147.725,172.500,49.017,159.814
C08170=1023.509,380.194,-147.766,172.509,49.017,159.816
C08171=1023.518,380.441,-147.808,172.518,49.018,159.818
C08172=1023.528,380.694,-147.850,172.528,49.018,159.819
C08173=1023.537,380.948,-147.892,172.536,49.019,159.821
C08174=1023.545,381.201,-147.936,172.546,49.020,159.822
C08175=1023.555,381.454,-147.978,172.555,49.021,159.824
C08176=1023.564,381.701,-148.020,172.565,49.021,159.826
C08177=1023.573,381.947,-148.061,172.574,49.022,159.827
C08178=1023.582,382.194,-148.103,172.584,49.023,159.829
C08179=1023.591,382.441,-148.144,172.593,49.023,159.830
C08180=1023.600,382.687,-148.186,172.601,49.024,159.832
C08181=1023.608,382.932,-148.228,172.611,49.024,159.833
C08182=1023.618,383.179,-148.270,172.620,49.025,159.835
C08183=1023.627,383.425,-148.311,172.630,49.026,159.837
C08184=1023.636,383.671,-148.353,172.639,49.027,159.838
C08185=1023.645,383.918,-148.394,172.649,49.027,159.840
C08186=1023.654,384.164,-148.436,172.658,49.029,159.842
C08187=1023.663,384.411,-148.478,172.668,49.029,159.843
C08188=1023.672,384.657,-148.520,172.677,49.030,159.845
C08189=1023.681,384.903,-148.562,172.687,49.031,159.847
C08190=1023.690,385.149,-148.604,172.695,49.032,159.848
C08191=1023.700,385.395,-148.645,172.706,49.033,159.850
C08192=1023.710,385.642,-148.688,172.714,49.033,159.852
C08193=1023.719,385.888,-148.729,172.725,49.034,159.853
C08194=1023.728,386.134,-148.772,172.733,49.035,159.855
C08195=1023.736,386.380,-148.814,172.744,49.036,159.857
C08196=1023.745,386.626,-148.857,172.753,49.036,159.858
C08197=1023.755,386.873,-148.899,172.763,49.038,159.860
C08198=1023.764,387.119,-148.941,172.773,49.039,159.862
C08199=1023.773,387.365,-148.984,172.782,49.040,159.864
C08200=1023.782,387.611,-149.025,172.792,49.040,159.865
C08201=1023.792,387.857,-149.068,172.802,49.041,159.867
C08202=1023.801,388.103,-149.110,172.811,49.043,159.869
C08203=1023.810,388.349,-149.154,172.821,49.044,159.871
C08204=1023.820,388.596,-149.196,172.831,49.045,159.872
C08205=1023.829,388.842,-149.238,172.840,49.046,159.874
C08206=1023.839,389.088,-149.281,172.851,49.047,159.876
C08207=1023.848,389.334,-149.323,172.861,49.048,159.878
C08208=1023.856,389.580,-149.366,172.870,49.049,159.880
C08209=1023.866,389.827,-149.409,172.880,49.050,159.881
C08210=1023.876,390.072,-149.452,172.890,49.051,159.883
C08211=1023.885,390.319,-149.496,172.899,49.052,159.885
C08212=1023.894,390.564,-149.538,172.910,49.053,159.887
C08213=1023.904,390.811,-149.581,172.920,49.054,159.889
C08214=1023.912,391.057,-149.624,172.930,49.056,159.891
C08215=1023.922,391.303,-149.667,172.940,49.057,159.892
C08216=1023.932,391.548,-149.710,172.950,49.058,159.894
C08217=1023.942,391.795,-149.753,172.960,49.060,159.896
C08218=1023.950,392.041,-149.796,172.970,49.061,159.898
C08219=1023.960,392.287,-149.839,172.980,49.062,159.900
C08220=1023.970,392.533,-149.882,172.991,49.063,159.902
C08221=1023.979,392.779,-149.926,173.001,49.064,159.904
C08222=1023.989,393.025,-149.969,173.011,49.066,159.906
C08223=1023.999,393.271,-150.012,173.021,49.067,159.907
C08224=1024.007,393.517,-150.055,173.031,49.068,159.909
C08225=1024.018,393.763,-150.099,173.041,49.069,159.911
C08226=1024.027,394.009,-150.143,173.052,49.071,159.913
C08227=1024.037,394.255,-150.186,173.063,49.072,159.915
C08228=1024.046,394.501,-150.229,173.073,49.073,159.917
C08229=1024.056,394.747,-150.273,173.083,49.075,159.919
C08230=1024.065,394.993,-150.317,173.094,49.076,159.921
C08231=1024.075,395.239,-150.360,173.104,49.078,159.923
C08232=1024.086,395.529,-150.412,173.116,49.080,159.926
C08233=1024.098,395.820,-150.463,173.129,49.081,159.928
C08234=1024.109,396.109,-150.515,173.141,49.083,159.930
C08235=1024.120,396.399,-150.567,173.154,49.085,159.933
C08236=1024.131,396.645,-150.610,173.164,49.086,159.935
C08237=1024.140,396.891,-150.654,173.175,49.088,159.937
C08238=1024.150,397.137,-150.698,173.185,49.089,159.939
C08239=1024.160,397.383,-150.743,173.196,49.091,159.941
C08240=1024.170,397.629,-150.786,173.207,49.093,159.943
C08241=1024.179,397.875,-150.830,173.217,49.094,159.945
C08242=1024.189,398.121,-150.874,173.228,49.096,159.947
C08243=1024.200,398.367,-150.919,173.239,49.097,159.949
C08244=1024.209,398.613,-150.963,173.250,49.098,159.951
C08245=1024.220,398.858,-151.007,173.261,49.100,159.953
C08246=1024.229,399.104,-151.051,173.271,49.102,159.955
C08247=1024.239,399.350,-151.096,173.282,49.104,159.958
C08248=1024.249,399.596,-151.140,173.294,49.105,159.960
C08249=1024.259,399.841,-151.185,173.304,49.107,159.962
C08250=1024.268,400.087,-151.229,173.315,49.109,159.964
C08251=1024.279,400.333,-151.273,173.326,49.110,159.966
C08252=1024.289,400.579,-151.318,173.338,49.112,159.968
C08253=1024.299,400.824,-151.363,173.348,49.114,159.971
C08254=1024.308,401.070,-151.407,173.359,49.116,159.973
C08255=1024.319,401.316,-151.452,173.371,49.117,159.975
C08256=1024.329,401.562,-151.496,173.382,49.119,159.977
C08257=1024.338,401.807,-151.541,173.393,49.121,159.979
C08258=1024.349,402.053,-151.587,173.404,49.123,159.981
C08259=1024.358,402.299,-151.631,173.415,49.125,159.984
C08260=1024.368,402.544,-151.676,173.426,49.127,159.986
C08261=1024.379,402.790,-151.722,173.438,49.128,159.988
C08262=1024.389,403.036,-151.767,173.449,49.131,159.990
C08263=1024.400,403.281,-151.811,173.460,49.133,159.993
C08264=1024.409,403.527,-151.856,173.472,49.134,159.995
C08265=1024.419,403.772,-151.902,173.483,49.136,159.997
C08266=1024.430,404.018,-151.947,173.494,49.138,160.000
C08267=1024.439,404.264,-151.992,173.505,49.140,160.002
C08268=1024.450,404.509,-152.038,173.518,49.142,160.004
C08269=1024.460,404.755,-152.083,173.528,49.144,160.007
C08270=1024.470,405.001,-152.128,173.540,49.146,160.009
C08271=1024.481,405.247,-152.174,173.552,49.148,160.011
C08272=1024.491,405.491,-152.219,173.564,49.150,160.014
C08273=1024.502,405.737,-152.264,173.575,49.152,160.016
C08274=1024.512,405.983,-152.310,173.586,49.154,160.018
C08275=1024.523,406.229,-152.355,173.599,49.156,160.021
C08276=1024.533,406.474,-152.400,173.610,49.158,160.023
C08277=1024.543,406.720,-152.446,173.622,49.161,160.026
C08278=1024.554,406.965,-152.492,173.634,49.162,160.028
C08279=1024.564,407.211,-152.537,173.646,49.165,160.030
C08280=1024.575,407.457,-152.583,173.657,49.167,160.033
C08281=1024.585,407.702,-152.629,173.669,49.169,160.035
C08282=1024.595,407.948,-152.675,173.681,49.171,160.038
C08283=1024.606,408.193,-152.721,173.694,49.174,160.040
C08284=1024.617,408.438,-152.766,173.706,49.176,160.043
C08285=1024.628,408.684,-152.812,173.717,49.178,160.045
C08286=1024.639,408.930,-152.858,173.729,49.180,160.047
C08287=1024.649,409.175,-152.904,173.741,49.182,160.050
C08288=1024.660,409.421,-152.950,173.754,49.185,160.053
C08289=1024.671,409.666,-152.996,173.766,49.187,160.055
C08290=1024.682,409.911,-153.042,173.778,49.189,160.058
C08291=1024.691,410.157,-153.089,173.790,49.191,160.060
C08292=1024.705,410.471,-153.148,173.806,49.195,160.063
C08293=1024.719,410.782,-153.207,173.821,49.198,160.067
C08294=1024.733,411.096,-153.266,173.837,49.201,160.070
C08295=1024.746,411.408,-153.325,173.852,49.204,160.073
C08296=1024.757,411.654,-153.373,173.865,49.206,160.076
C08297=1024.768,411.899,-153.419,173.877,49.209,160.078
C08298=1024.779,412.145,-153.465,173.890,49.211,160.081
C08299=1024.790,412.390,-153.512,173.902,49.214,160.084
C08300=1024.801,412.635,-153.559,173.915,49.216,160.086
C08301=1024.811,412.881,-153.606,173.927,49.219,160.089
C08302=1024.822,413.126,-153.653,173.941,49.221,160.092
C08303=1024.834,413.371,-153.700,173.953,49.224,160.095
C08304=1024.845,413.616,-153.746,173.966,49.226,160.097
C08305=1024.855,413.862,-153.793,173.978,49.229,160.100
C08306=1024.866,414.107,-153.840,173.991,49.231,160.103
C08307=1024.877,414.352,-153.887,174.005,49.234,160.105
C08308=1024.889,414.598,-153.934,174.017,49.237,160.108
C08309=1024.899,414.843,-153.981,174.030,49.239,160.111
C08310=1024.911,415.089,-154.028,174.042,49.242,160.113
C08311=1024.922,415.334,-154.076,174.056,49.244,160.116
C08312=1024.933,415.579,-154.123,174.069,49.247,160.119
C08313=1024.944,415.825,-154.170,174.081,49.250,160.122
C08314=1024.956,416.070,-154.218,174.095,49.252,160.125
C08315=1024.966,416.315,-154.265,174.108,49.255,160.127
C08316=1024.978,416.560,-154.313,174.120,49.258,160.130
C08317=1024.989,416.806,-154.360,174.134,49.261,160.133
C08318=1025.000,417.051,-154.408,174.147,49.264,160.136
C08319=1025.011,417.296,-154.456,174.161,49.266,160.139
C08320=1025.023,417.541,-154.504,174.174,49.269,160.142
C08321=1025.033,417.786,-154.551,174.187,49.272,160.145
C08322=1025.045,418.031,-154.599,174.200,49.275,160.148
C08323=1025.056,418.277,-154.647,174.214,49.278,160.151
C08324=1025.068,418.522,-154.695,174.227,49.281,160.153
C08325=1025.079,418.767,-154.743,174.241,49.284,160.156
C08326=1025.091,419.012,-154.791,174.255,49.286,160.159
C08327=1025.102,419.258,-154.839,174.268,49.289,160.162
C08328=1025.114,419.503,-154.887,174.282,49.292,160.165
C08329=1025.125,419.748,-154.935,174.296,49.295,160.168
C08330=1025.137,419.992,-154.983,174.309,49.298,160.171
C08331=1025.148,420.238,-155.032,174.323,49.301,160.174
C08332=1025.160,420.483,-155.079,174.337,49.304,160.177
C08333=1025.171,420.728,-155.128,174.351,49.307,160.180
C08334=1025.183,420.973,-155.176,174.364,49.310,160.183
C08335=1025.194,421.218,-155.224,174.378,49.313,160.186
C08336=1025.207,421.462,-155.273,174.392,49.317,160.190
C08337=1025.218,421.709,-155.321,174.406,49.320,160.193
C08338=1025.230,421.953,-155.370,174.420,49.322,160.196
C08339=1025.242,422.198,-155.419,174.435,49.326,160.199
C08340=1025.253,422.444,-155.468,174.449,49.329,160.202
C08341=1025.265,422.689,-155.517,174.463,49.332,160.205
C08342=1025.277,422.933,-155.565,174.477,49.335,160.208
C08343=1025.288,423.178,-155.614,174.492,49.339,160.212
C08344=1025.300,423.423,-155.663,174.506,49.341,160.215
C08345=1025.313,423.668,-155.712,174.520,49.345,160.218
C08346=1025.325,423.913,-155.761,174.534,49.348,160.221
C08347=1025.336,424.158,-155.810,174.548,49.351,160.224
C08348=1025.347,424.402,-155.859,174.563,49.354,160.227
C08349=1025.360,424.648,-155.908,174.577,49.358,160.231
C08350=1025.372,424.892,-155.958,174.592,49.361,160.234
C08351=1025.384,425.137,-156.007,174.607,49.364,160.237
C08352=1025.398,425.404,-156.061,174.623,49.368,160.241
C08353=1025.411,425.672,-156.115,174.639,49.372,160.245
C08354=1025.423,425.938,-156.169,174.655,49.376,160.248
C08355=1025.437,426.205,-156.222,174.670,49.379,160.252
C08356=1025.449,426.451,-156.272,174.686,49.382,160.255
C08357=1025.461,426.696,-156.322,174.701,49.386,160.258
C08358=1025.473,426.940,-156.371,174.715,49.390,160.262
C08359=1025.485,427.185,-156.422,174.731,49.393,160.265
C08360=1025.498,427.429,-156.472,174.745,49.397,160.268
C08361=1025.510,427.675,-156.521,174.761,49.400,160.272
C08362=1025.521,427.919,-156.571,174.776,49.404,160.276
C08363=1025.534,428.164,-156.621,174.791,49.407,160.279
C08364=1025.549,428.465,-156.683,174.810,49.412,160.283
C08365=1025.564,428.766,-156.744,174.829,49.416,160.288
C08366=1025.580,429.068,-156.807,174.848,49.421,160.292
C08367=1025.595,429.368,-156.868,174.867,49.425,160.296
C08368=1025.608,429.613,-156.918,174.883,49.429,160.300
C08369=1025.620,429.858,-156.968,174.897,49.433,160.303
C08370=1025.632,430.102,-157.019,174.913,49.436,160.307
C08371=1025.645,430.347,-157.069,174.929,49.440,160.310
C08372=1025.657,430.591,-157.120,174.945,49.443,160.314
C08373=1025.670,430.836,-157.170,174.959,49.447,160.317
C08374=1025.682,431.080,-157.221,174.976,49.451,160.321
C08375=1025.696,431.325,-157.272,174.991,49.455,160.325
C08376=1025.708,431.570,-157.322,175.008,49.459,160.328
C08377=1025.720,431.814,-157.373,175.023,49.462,160.332
C08378=1025.734,432.059,-157.424,175.040,49.466,160.336
C08379=1025.746,432.303,-157.475,175.055,49.470,160.339
C08380=1025.759,432.548,-157.525,175.071,49.474,160.343
C08381=1025.772,432.793,-157.576,175.088,49.478,160.347
C08382=1025.784,433.037,-157.627,175.104,49.482,160.351
C08383=1025.798,433.282,-157.679,175.120,49.486,160.354
C08384=1025.811,433.526,-157.730,175.137,49.490,160.358
C08385=1025.824,433.771,-157.781,175.153,49.494,160.362
C08386=1025.836,434.015,-157.832,175.170,49.498,160.366
C08387=1025.850,434.259,-157.884,175.186,49.502,160.370
C08388=1025.863,434.503,-157.935,175.203,49.505,160.373
C08389=1025.875,434.748,-157.987,175.219,49.509,160.377
C08390=1025.889,434.993,-158.038,175.236,49.514,160.381
C08391=1025.902,435.237,-158.090,175.253,49.517,160.385
C08392=1025.915,435.481,-158.141,175.269,49.522,160.389
C08393=1025.928,435.726,-158.193,175.285,49.526,160.393
C08394=1025.941,435.970,-158.245,175.303,49.530,160.397
C08395=1025.954,436.214,-158.297,175.320,49.535,160.401
C08396=1025.968,436.458,-158.349,175.337,49.538,160.405
C08397=1025.981,436.702,-158.401,175.353,49.543,160.409
C08398=1025.995,436.947,-158.453,175.371,49.547,160.413
C08399=1026.007,437.191,-158.505,175.388,49.551,160.417
C08400=1026.021,437.435,-158.557,175.405,49.555,160.421
C08401=1026.034,437.680,-158.609,175.423,49.560,160.425
C08402=1026.048,437.923,-158.661,175.440,49.564,160.429
C08403=1026.061,438.168,-158.714,175.458,49.568,160.433
C08404=1026.075,438.412,-158.766,175.474,49.572,160.437
C08405=1026.088,438.656,-158.818,175.492,49.577,160.441
C08406=1026.101,438.901,-158.871,175.510,49.581,160.446
C08407=1026.115,439.144,-158.923,175.528,49.586,160.450
C08408=1026.129,439.388,-158.976,175.545,49.590,160.454
C08409=1026.142,439.633,-159.029,175.563,49.594,160.458
C08410=1026.156,439.877,-159.082,175.581,49.598,160.462
C08411=1026.170,440.120,-159.134,175.599,49.603,160.467
C08412=1026.182,440.340,-159.182,175.615,49.607,160.470
C08413=1026.194,440.560,-159.229,175.631,49.611,160.474
C08414=1026.207,440.780,-159.277,175.648,49.615,160.478
C08415=1026.220,440.999,-159.324,175.664,49.619,160.482
C08416=1026.232,441.218,-159.373,175.680,49.623,160.486
C08417=1026.245,441.438,-159.421,175.697,49.627,160.490
C08418=1026.257,441.658,-159.468,175.713,49.631,160.494
C08419=1026.270,441.877,-159.516,175.729,49.635,160.498
C08420=1026.284,442.120,-159.569,175.748,49.640,160.502
C08421=1026.298,442.363,-159.622,175.766,49.645,160.506
C08422=1026.313,442.607,-159.676,175.785,49.649,160.511
C08423=1026.326,442.851,-159.728,175.803,49.654,160.515
C08424=1026.341,443.094,-159.780,175.822,49.658,160.520
C08425=1026.357,443.337,-159.833,175.841,49.662,160.524
C08426=1026.373,443.581,-159.885,175.859,49.667,160.528
C08427=1026.389,443.825,-159.935,175.878,49.671,160.533
C08428=1026.406,444.068,-159.986,175.897,49.675,160.537
C08429=1026.423,444.312,-160.036,175.917,49.679,160.542
C08430=1026.442,444.556,-160.087,175.936,49.683,160.546
C08431=1026.460,444.800,-160.137,175.955,49.687,160.550
C08432=1026.478,445.044,-160.185,175.975,49.691,160.555
C08433=1026.497,445.288,-160.234,175.994,49.695,160.559
C08434=1026.517,445.532,-160.283,176.013,49.699,160.563
C08435=1026.537,445.776,-160.331,176.033,49.702,160.568
C08436=1026.557,446.021,-160.379,176.053,49.706,160.572
C08437=1026.578,446.265,-160.426,176.073,49.709,160.576
C08438=1026.600,446.510,-160.473,176.093,49.713,160.581
C08439=1026.621,446.754,-160.519,176.112,49.716,160.585
C08440=1026.644,446.998,-160.566,176.132,49.720,160.589
C08441=1026.667,447.243,-160.611,176.153,49.723,160.594
C08442=1026.690,447.488,-160.656,176.173,49.726,160.598
C08443=1026.714,447.733,-160.702,176.193,49.729,160.602
C08444=1026.738,447.978,-160.746,176.213,49.733,160.607
C08445=1026.763,448.223,-160.790,176.234,49.736,160.611
C08446=1026.787,448.467,-160.834,176.254,49.738,160.615
C08447=1026.813,448.713,-160.877,176.275,49.742,160.620
C08448=1026.839,448.958,-160.920,176.295,49.744,160.624
C08449=1026.866,449.203,-160.963,176.316,49.747,160.628
C08450=1026.893,449.448,-161.005,176.338,49.750,160.633
C08451=1026.920,449.693,-161.047,176.358,49.753,160.637
C08452=1026.948,449.938,-161.087,176.380,49.755,160.641
C08453=1026.976,450.184,-161.129,176.400,49.758,160.645
C08454=1027.004,450.430,-161.170,176.422,49.760,160.650
C08455=1027.034,450.675,-161.210,176.443,49.762,160.654
C08456=1027.064,450.920,-161.250,176.465,49.765,160.658
C08457=1027.093,451.166,-161.289,176.486,49.767,160.663
C08458=1027.124,451.411,-161.329,176.508,49.769,160.667
C08459=1027.156,451.656,-161.367,176.530,49.772,160.671
C08460=1027.187,451.902,-161.405,176.552,49.774,160.676
C08461=1027.219,452.148,-161.443,176.573,49.776,160.680
C08462=1027.251,452.394,-161.481,176.595,49.778,160.684
C08463=1027.284,452.638,-161.518,176.618,49.780,160.688
C08464=1027.317,452.885,-161.555,176.639,49.782,160.693
C08465=1027.351,453.131,-161.591,176.662,49.784,160.697
C08466=1027.385,453.376,-161.627,176.684,49.786,160.701
C08467=1027.420,453.622,-161.662,176.707,49.788,160.706
C08468=1027.456,453.868,-161.697,176.730,49.789,160.710
C08469=1027.491,454.114,-161.732,176.752,49.791,160.714
C08470=1027.528,454.359,-161.766,176.775,49.792,160.718
C08471=1027.564,454.605,-161.800,176.798,49.794,160.723
C08472=1027.290,454.683,-162.139,176.801,49.854,160.742
C08473=1027.254,454.438,-162.104,176.778,49.853,160.738
C08474=1027.218,454.192,-162.070,176.755,49.850,160.733
C08475=1027.181,453.946,-162.035,176.732,49.849,160.729
C08476=1027.146,453.700,-162.001,176.709,49.847,160.725
C08477=1027.112,453.455,-161.965,176.687,49.846,160.721
C08478=1027.077,453.209,-161.930,176.665,49.844,160.717
C08479=1027.043,452.963,-161.893,176.642,49.842,160.712
C08480=1027.010,452.717,-161.857,176.620,49.840,160.708
C08481=1026.977,452.472,-161.820,176.597,49.839,160.704
C08482=1026.944,452.226,-161.783,176.575,49.837,160.699
C08483=1026.911,451.980,-161.745,176.554,49.835,160.695
C08484=1026.880,451.735,-161.707,176.531,49.833,160.691
C08485=1026.849,451.489,-161.668,176.510,49.831,160.687
C08486=1026.818,451.243,-161.629,176.487,49.829,160.682
C08487=1026.788,450.998,-161.590,176.466,49.826,160.678
C08488=1026.757,450.752,-161.550,176.445,49.824,160.674
C08489=1026.729,450.507,-161.510,176.423,49.822,160.669
C08490=1026.700,450.262,-161.470,176.401,49.819,160.665
C08491=1026.671,450.016,-161.429,176.381,49.817,160.661
C08492=1026.643,449.771,-161.388,176.360,49.815,160.657
C08493=1026.615,449.525,-161.346,176.338,49.812,160.652
C08494=1026.588,449.281,-161.304,176.317,49.809,160.648
C08495=1026.561,449.036,-161.261,176.297,49.807,160.644
C08496=1026.536,448.790,-161.219,176.275,49.804,160.639
C08497=1026.510,448.545,-161.176,176.255,49.801,160.635
C08498=1026.484,448.300,-161.132,176.234,49.798,160.631
C08499=1026.460,448.056,-161.089,176.213,49.796,160.626
C08500=1026.435,447.811,-161.044,176.193,49.792,160.622
C08501=1026.411,447.566,-161.000,176.173,49.789,160.618
C08502=1026.388,447.321,-160.954,176.152,49.786,160.613
C08503=1026.365,447.076,-160.908,176.133,49.783,160.609
C08504=1026.343,446.832,-160.862,176.112,49.780,160.605
C08505=1026.321,446.587,-160.816,176.092,49.777,160.601
C08506=1026.299,446.343,-160.769,176.072,49.773,160.596
C08507=1026.278,446.099,-160.722,176.053,49.770,160.592
C08508=1026.257,445.854,-160.674,176.033,49.766,160.588
C08509=1026.236,445.609,-160.627,176.013,49.763,160.583
C08510=1026.218,445.365,-160.579,175.993,49.759,160.579
C08511=1026.198,445.122,-160.530,175.973,49.755,160.574
C08512=1026.178,444.878,-160.481,175.955,49.752,160.570
C08513=1026.160,444.633,-160.432,175.935,49.748,160.566
C08514=1026.143,444.389,-160.382,175.916,49.744,160.562
C08515=1026.125,444.145,-160.331,175.897,49.740,160.557
C08516=1026.108,443.902,-160.281,175.878,49.736,160.553
C08517=1026.092,443.658,-160.230,175.858,49.732,160.548
C08518=1026.076,443.415,-160.178,175.840,49.728,160.544
C08519=1026.060,443.171,-160.127,175.821,49.724,160.540
C08520=1026.044,442.928,-160.075,175.802,49.720,160.535
C08521=1026.029,442.684,-160.022,175.783,49.715,160.531
C08522=1026.015,442.441,-159.970,175.765,49.710,160.526
C08523=1026.001,442.198,-159.916,175.746,49.706,160.522
C08524=1025.987,441.955,-159.863,175.728,49.702,160.518
C08525=1025.975,441.739,-159.816,175.712,49.698,160.514
C08526=1025.962,441.524,-159.770,175.695,49.694,160.510
C08527=1025.950,441.308,-159.723,175.679,49.690,160.506
C08528=1025.937,441.092,-159.676,175.663,49.686,160.502
C08529=1025.925,440.877,-159.628,175.648,49.682,160.499
C08530=1025.913,440.662,-159.582,175.631,49.678,160.495
C08531=1025.901,440.446,-159.535,175.615,49.674,160.491
C08532=1025.888,440.231,-159.489,175.599,49.670,160.487
C08533=1025.875,439.987,-159.436,175.581,49.666,160.483
C08534=1025.861,439.742,-159.383,175.563,49.662,160.479
C08535=1025.847,439.499,-159.330,175.546,49.658,160.475
C08536=1025.834,439.255,-159.277,175.528,49.653,160.470
C08537=1025.820,439.011,-159.225,175.510,49.649,160.466
C08538=1025.807,438.767,-159.173,175.492,49.645,160.462
C08539=1025.794,438.522,-159.120,175.475,49.640,160.458
C08540=1025.780,438.279,-159.067,175.457,49.636,160.454
C08541=1025.766,438.034,-159.015,175.440,49.632,160.450
C08542=1025.752,437.789,-158.963,175.423,49.628,160.446
C08543=1025.739,437.545,-158.910,175.405,49.624,160.442
C08544=1025.726,437.301,-158.858,175.388,49.620,160.437
C08545=1025.712,437.057,-158.806,175.370,49.616,160.433
C08546=1025.699,436.813,-158.754,175.354,49.611,160.429
C08547=1025.686,436.569,-158.702,175.336,49.608,160.425
C08548=1025.673,436.324,-158.650,175.319,49.603,160.421
C08549=1025.659,436.080,-158.598,175.302,49.599,160.417
C08550=1025.646,435.836,-158.547,175.285,49.595,160.414
C08551=1025.633,435.592,-158.496,175.268,49.591,160.409
C08552=1025.620,435.347,-158.443,175.251,49.587,160.406
C08553=1025.607,435.103,-158.391,175.235,49.583,160.402
C08554=1025.594,434.858,-158.340,175.218,49.579,160.398
C08555=1025.581,434.614,-158.289,175.201,49.575,160.394
C08556=1025.568,434.369,-158.238,175.185,49.571,160.390
C08557=1025.555,434.126,-158.186,175.168,49.568,160.386
C08558=1025.542,433.881,-158.134,175.152,49.564,160.383
C08559=1025.529,433.636,-158.083,175.136,49.560,160.379
C08560=1025.516,433.392,-158.032,175.119,49.556,160.375
C08561=1025.503,433.148,-157.981,175.102,49.552,160.371
C08562=1025.490,432.903,-157.930,175.086,49.549,160.368
C08563=1025.478,432.659,-157.879,175.070,49.544,160.364
C08564=1025.464,432.414,-157.828,175.054,49.540,160.360
C08565=1025.452,432.170,-157.777,175.038,49.537,160.356
C08566=1025.439,431.924,-157.726,175.022,49.533,160.353
C08567=1025.426,431.680,-157.675,175.006,49.530,160.349
C08568=1025.414,431.436,-157.625,174.990,49.525,160.345
C08569=1025.401,431.192,-157.574,174.974,49.522,160.342
C08570=1025.387,430.946,-157.524,174.958,49.518,160.338
C08571=1025.375,430.702,-157.473,174.943,49.515,160.335
C08572=1025.362,430.457,-157.423,174.926,49.511,160.331
C08573=1025.350,430.213,-157.372,174.911,49.507,160.327
C08574=1025.337,429.968,-157.322,174.895,49.504,160.324
C08575=1025.325,429.724,-157.271,174.880,49.500,160.320
C08576=1025.313,429.479,-157.221,174.864,49.497,160.317
C08577=1025.300,429.234,-157.171,174.849,49.494,160.313
C08578=1025.288,428.990,-157.121,174.833,49.490,160.310
C08579=1025.275,428.745,-157.070,174.818,49.486,160.306
C08580=1025.263,428.501,-157.020,174.802,49.483,160.303
C08581=1025.251,428.256,-156.970,174.787,49.480,160.299
C08582=1025.238,428.011,-156.920,174.772,49.476,160.296
C08583=1025.226,427.766,-156.870,174.756,49.472,160.292
C08584=1025.214,427.521,-156.820,174.742,49.469,160.289
C08585=1025.201,427.278,-156.771,174.726,49.465,160.285
C08586=1025.189,427.032,-156.721,174.712,49.462,160.282
C08587=1025.177,426.787,-156.671,174.696,49.459,160.279
C08588=1025.165,426.542,-156.621,174.681,49.455,160.275
C08589=1025.149,426.217,-156.555,174.662,49.451,160.271
C08590=1025.133,425.891,-156.489,174.642,49.446,160.266
C08591=1025.117,425.565,-156.423,174.623,49.442,160.262
C08592=1025.101,425.239,-156.358,174.603,49.438,160.258
C08593=1025.089,424.994,-156.309,174.588,49.434,160.254
C08594=1025.077,424.748,-156.259,174.573,49.431,160.251
C08595=1025.065,424.505,-156.210,174.559,49.428,160.248
C08596=1025.053,424.259,-156.161,174.545,49.425,160.245
C08597=1025.041,424.014,-156.112,174.530,49.421,160.241
C08598=1025.029,423.769,-156.062,174.516,49.418,160.238
C08599=1025.017,423.525,-156.014,174.501,49.416,160.235
C08600=1025.005,423.279,-155.965,174.486,49.412,160.232
C08601=1024.994,423.034,-155.916,174.472,49.409,160.229
C08602=1024.982,422.790,-155.867,174.458,49.406,160.225
C08603=1024.970,422.545,-155.818,174.444,49.403,160.222
C08604=1024.958,422.299,-155.769,174.429,49.400,160.219
C08605=1024.941,421.925,-155.695,174.408,49.395,160.214
C08606=1024.923,421.551,-155.621,174.387,49.390,160.210
C08607=1024.905,421.176,-155.547,174.366,49.386,160.205
C08608=1024.887,420.802,-155.473,174.344,49.381,160.200
C08609=1024.875,420.557,-155.425,174.330,49.378,160.197
C08610=1024.864,420.313,-155.376,174.316,49.375,160.194
C08611=1024.852,420.068,-155.328,174.302,49.372,160.191
C08612=1024.841,419.822,-155.280,174.289,49.370,160.188
C08613=1024.829,419.577,-155.232,174.275,49.367,160.185
C08614=1024.818,419.332,-155.184,174.262,49.364,160.182
C08615=1024.806,419.087,-155.136,174.247,49.361,160.179
C08616=1024.795,418.841,-155.088,174.234,49.359,160.177
C08617=1024.783,418.596,-155.040,174.221,49.355,160.174
C08618=1024.772,418.351,-154.992,174.207,49.353,160.171
C08619=1024.760,418.106,-154.944,174.193,49.350,160.168
C08620=1024.749,417.861,-154.897,174.180,49.347,160.165
C08621=1024.738,417.616,-154.849,174.166,49.345,160.162
C08622=1024.727,417.371,-154.801,174.154,49.342,160.159
C08623=1024.715,417.125,-154.754,174.140,49.339,160.156
C08624=1024.704,416.880,-154.706,174.127,49.336,160.153
C08625=1024.693,416.635,-154.658,174.113,49.334,160.150
C08626=1024.682,416.389,-154.610,174.101,49.331,160.148
C08627=1024.671,416.145,-154.563,174.087,49.329,160.145
C08628=1024.660,415.899,-154.515,174.074,49.325,160.142
C08629=1024.648,415.654,-154.468,174.061,49.323,160.139
C08630=1024.637,415.409,-154.421,174.048,49.320,160.136
C08631=1024.626,415.163,-154.374,174.035,49.318,160.134
C08632=1024.614,414.918,-154.326,174.022,49.316,160.131
C08633=1024.604,414.673,-154.279,174.009,49.313,160.128
C08634=1024.592,414.427,-154.232,173.996,49.310,160.125
C08635=1024.582,414.182,-154.185,173.983,49.308,160.123
C08636=1024.570,413.936,-154.138,173.971,49.306,160.120
C08637=1024.559,413.691,-154.091,173.958,49.303,160.117
C08638=1024.548,413.446,-154.044,173.945,49.300,160.115
C08639=1024.538,413.200,-153.997,173.932,49.298,160.112
C08640=1024.527,412.955,-153.951,173.919,49.296,160.109
C08641=1024.515,412.710,-153.904,173.907,49.293,160.107
C08642=1024.504,412.465,-153.857,173.894,49.291,160.104
C08643=1024.494,412.219,-153.810,173.882,49.288,160.101
C08644=1024.483,411.974,-153.764,173.869,49.286,160.099
C08645=1024.473,411.758,-153.723,173.858,49.284,160.096
C08646=1024.464,411.542,-153.681,173.848,49.282,160.094
C08647=1024.454,411.327,-153.641,173.837,49.280,160.092
C08648=1024.445,411.112,-153.600,173.826,49.278,160.090
C08649=1024.436,410.896,-153.559,173.815,49.276,160.087
C08650=1024.426,410.681,-153.518,173.804,49.274,160.085
C08651=1024.416,410.465,-153.478,173.793,49.272,160.083
C08652=1024.408,410.249,-153.437,173.782,49.270,160.081
C08653=1024.397,410.004,-153.391,173.770,49.268,160.078
C08654=1024.386,409.759,-153.344,173.757,49.265,160.075
C08655=1024.375,409.513,-153.298,173.745,49.263,160.073
C08656=1024.365,409.267,-153.252,173.733,49.261,160.070
C08657=1024.354,409.022,-153.207,173.722,49.258,160.068
C08658=1024.343,408.776,-153.161,173.709,49.256,160.065
C08659=1024.333,408.531,-153.114,173.697,49.255,160.063
C08660=1024.322,408.286,-153.068,173.685,49.252,160.060
C08661=1024.312,408.039,-153.023,173.673,49.250,160.058
C08662=1024.301,407.794,-152.977,173.661,49.248,160.056
C08663=1024.290,407.548,-152.931,173.649,49.246,160.053
C08664=1024.280,407.303,-152.886,173.638,49.244,160.051
C08665=1024.269,407.058,-152.840,173.625,49.242,160.048
C08666=1024.258,406.812,-152.794,173.614,49.240,160.046
C08667=1024.248,406.566,-152.749,173.601,49.238,160.043
C08668=1024.237,406.321,-152.703,173.590,49.236,160.041
C08669=1024.227,406.076,-152.658,173.578,49.234,160.039
C08670=1024.217,405.830,-152.613,173.566,49.232,160.036
C08671=1024.206,405.584,-152.567,173.555,49.230,160.034
C08672=1024.196,405.339,-152.521,173.543,49.228,160.032
C08673=1024.186,405.093,-152.476,173.531,49.226,160.029
C08674=1024.175,404.847,-152.430,173.520,49.224,160.027
C08675=1024.165,404.602,-152.386,173.508,49.222,160.025
C08676=1024.155,404.356,-152.341,173.496,49.221,160.022
C08677=1024.145,404.111,-152.295,173.485,49.219,160.020
C08678=1024.134,403.865,-152.250,173.474,49.217,160.018
C08679=1024.125,403.619,-152.205,173.463,49.215,160.016
C08680=1024.114,403.374,-152.159,173.451,49.213,160.013
C08681=1024.104,403.128,-152.114,173.440,49.211,160.011
C08682=1024.094,402.882,-152.069,173.428,49.209,160.009
C08683=1024.084,402.636,-152.024,173.417,49.207,160.006
C08684=1024.074,402.391,-151.980,173.405,49.206,160.004
C08685=1024.064,402.145,-151.935,173.395,49.204,160.002
C08686=1024.054,401.899,-151.890,173.384,49.202,160.000
C08687=1024.044,401.654,-151.845,173.372,49.200,159.997
C08688=1024.034,401.408,-151.800,173.361,49.198,159.995
C08689=1024.024,401.162,-151.755,173.349,49.197,159.993
C08690=1024.014,400.917,-151.710,173.338,49.195,159.991
C08691=1024.004,400.672,-151.666,173.328,49.194,159.989
C08692=1023.994,400.425,-151.621,173.316,49.192,159.986
C08693=1023.984,400.179,-151.577,173.305,49.190,159.984
C08694=1023.974,399.934,-151.533,173.294,49.188,159.982
C08695=1023.964,399.688,-151.488,173.283,49.187,159.980
C08696=1023.955,399.442,-151.444,173.272,49.186,159.978
C08697=1023.944,399.197,-151.399,173.261,49.184,159.976
C08698=1023.934,398.950,-151.355,173.251,49.182,159.974
C08699=1023.924,398.705,-151.310,173.239,49.181,159.972
C08700=1023.914,398.459,-151.267,173.229,49.180,159.970
C08701=1023.905,398.213,-151.223,173.218,49.177,159.967
C08702=1023.895,397.967,-151.178,173.207,49.176,159.965
C08703=1023.885,397.721,-151.134,173.196,49.175,159.963
C08704=1023.876,397.475,-151.090,173.185,49.173,159.961
C08705=1023.865,397.230,-151.047,173.175,49.172,159.959
C08706=1023.856,396.984,-151.002,173.164,49.170,159.957
C08707=1023.846,396.738,-150.958,173.154,49.169,159.955
C08708=1023.836,396.492,-150.914,173.143,49.167,159.953
C08709=1023.824,396.200,-150.863,173.130,49.166,159.951
C08710=1023.813,395.907,-150.811,173.117,49.164,159.948
C08711=1023.801,395.614,-150.759,173.105,49.163,159.946
C08712=1023.790,395.322,-150.706,173.093,49.161,159.944
C08713=1023.780,395.075,-150.663,173.082,49.160,159.942
C08714=1023.770,394.829,-150.619,173.072,49.159,159.940
C08715=1023.761,394.584,-150.576,173.061,49.157,159.938
C08716=1023.752,394.338,-150.532,173.051,49.156,159.936
C08717=1023.741,394.092,-150.488,173.041,49.155,159.934
C08718=1023.732,393.846,-150.445,173.030,49.153,159.932
C08719=1023.723,393.600,-150.402,173.020,49.152,159.930
C08720=1023.713,393.354,-150.358,173.009,49.151,159.928
C08721=1023.703,393.108,-150.315,172.999,49.150,159.926
C08722=1023.694,392.863,-150.272,172.989,49.148,159.924
C08723=1023.685,392.616,-150.228,172.978,49.147,159.922
C08724=1023.675,392.370,-150.185,172.968,49.146,159.920
C08725=1023.665,392.124,-150.142,172.959,49.145,159.918
C08726=1023.656,391.878,-150.099,172.949,49.144,159.917
C08727=1023.647,391.632,-150.056,172.938,49.143,159.915
C08728=1023.637,391.386,-150.013,172.928,49.142,159.913
C08729=1023.627,391.140,-149.970,172.918,49.140,159.911
C08730=1023.619,390.894,-149.927,172.908,49.139,159.909
C08731=1023.608,390.648,-149.884,172.897,49.138,159.907
C08732=1023.599,390.402,-149.841,172.888,49.137,159.906
C08733=1023.590,390.155,-149.798,172.878,49.136,159.904
C08734=1023.581,389.909,-149.755,172.868,49.135,159.902
C08735=1023.572,389.664,-149.713,172.858,49.134,159.900
C08736=1023.562,389.417,-149.670,172.848,49.133,159.898
C08737=1023.553,389.171,-149.627,172.838,49.132,159.896
C08738=1023.543,388.925,-149.584,172.828,49.131,159.895
C08739=1023.534,388.679,-149.542,172.818,49.130,159.893
C08740=1023.525,388.433,-149.499,172.808,49.130,159.891
C08741=1023.515,388.187,-149.457,172.799,49.128,159.889
C08742=1023.507,387.940,-149.414,172.789,49.127,159.888
C08743=1023.498,387.694,-149.372,172.779,49.126,159.886
C08744=1023.488,387.448,-149.329,172.770,49.126,159.884
C08745=1023.479,387.202,-149.287,172.760,49.125,159.882
C08746=1023.470,386.956,-149.245,172.750,49.124,159.881
C08747=1023.460,386.710,-149.203,172.741,49.123,159.879
C08748=1023.451,386.463,-149.160,172.731,49.122,159.877
C08749=1023.442,386.217,-149.117,172.721,49.122,159.876
C08750=1023.433,385.971,-149.076,172.712,49.120,159.874
C08751=1023.424,385.725,-149.033,172.702,49.120,159.872
C08752=1023.415,385.479,-148.992,172.693,49.119,159.870
C08753=1023.405,385.232,-148.949,172.683,49.118,159.869
C08754=1023.396,384.986,-148.908,172.673,49.117,159.867
C08755=1023.387,384.740,-148.866,172.664,49.117,159.866
C08756=1023.378,384.493,-148.824,172.654,49.116,159.864
C08757=1023.369,384.248,-148.782,172.645,49.115,159.862
C08758=1023.360,384.001,-148.740,172.635,49.114,159.861
C08759=1023.351,383.755,-148.698,172.626,49.114,159.859
C08760=1023.342,383.508,-148.657,172.616,49.113,159.857
C08761=1023.332,383.262,-148.616,172.608,49.113,159.856
C08762=1023.323,383.016,-148.574,172.598,49.112,159.854
C08763=1023.314,382.770,-148.532,172.589,49.111,159.853
C08764=1023.305,382.523,-148.490,172.579,49.111,159.851
C08765=1023.296,382.277,-148.449,172.570,49.110,159.849
C08766=1023.288,382.031,-148.407,172.560,49.109,159.848
C08767=1023.279,381.784,-148.365,172.551,49.109,159.846
C08768=1023.269,381.538,-148.324,172.542,49.109,159.845
C08769=1023.260,381.282,-148.281,172.533,49.107,159.843
C08770=1023.251,381.026,-148.238,172.523,49.107,159.841
C08771=1023.242,380.771,-148.195,172.513,49.107,159.840
C08772=1023.233,380.515,-148.152,172.504,49.106,159.838
C08773=1023.224,380.268,-148.110,172.494,49.106,159.837
C08774=1023.215,380.022,-148.070,172.486,49.105,159.835
C08775=1023.206,379.775,-148.028,172.477,49.105,159.834
C08776=1023.197,379.529,-147.986,172.467,49.104,159.832
C08777=1023.189,379.283,-147.946,172.459,49.104,159.831
C08778=1023.180,379.036,-147.904,172.450,49.103,159.829
C08779=1023.171,378.789,-147.863,172.440,49.103,159.828
C08780=1023.163,378.544,-147.822,172.432,49.102,159.826
C08781=1023.154,378.297,-147.781,172.423,49.102,159.825
C08782=1023.145,378.051,-147.740,172.413,49.102,159.823
C08783=1023.137,377.804,-147.699,172.405,49.102,159.822
C08784=1023.128,377.558,-147.657,172.396,49.101,159.820
C08785=1023.119,377.311,-147.616,172.388,49.101,159.819
C08786=1023.111,377.065,-147.576,172.378,49.100,159.817
C08787=1023.102,376.818,-147.534,172.369,49.100,159.816
C08788=1023.093,376.572,-147.494,172.361,49.099,159.814
C08789=1023.085,376.325,-147.453,172.352,49.099,159.813
C08790=1023.076,376.078,-147.412,172.342,49.099,159.811
C08791=1023.067,375.832,-147.372,172.334,49.099,159.810
C08792=1023.059,375.585,-147.331,172.325,49.098,159.809
C08793=1023.050,375.340,-147.291,172.317,49.098,159.807
C08794=1023.041,375.093,-147.250,172.308,49.098,159.806
C08795=1023.033,374.847,-147.210,172.299,49.098,159.804
C08796=1023.024,374.600,-147.169,172.290,49.098,159.803
C08797=1023.015,374.354,-147.129,172.282,49.097,159.802
C08798=1023.007,374.107,-147.088,172.273,49.097,159.800
C08799=1022.998,373.861,-147.048,172.265,49.097,159.799
C08800=1022.989,373.613,-147.007,172.256,49.097,159.798
C08801=1022.981,373.367,-146.967,172.247,49.097,159.796
C08802=1022.973,373.121,-146.927,172.238,49.097,159.795
C08803=1022.963,372.874,-146.886,172.230,49.097,159.794
C08804=1022.956,372.627,-146.846,172.222,49.097,159.792
C08805=1022.947,372.381,-146.806,172.213,49.096,159.791
C08806=1022.939,372.134,-146.766,172.205,49.096,159.790
C08807=1022.930,371.887,-146.725,172.196,49.096,159.788
C08808=1022.922,371.641,-146.685,172.188,49.096,159.787
C08809=1022.913,371.394,-146.645,172.179,49.096,159.786
C08810=1022.905,371.148,-146.605,172.171,49.096,159.784
C08811=1022.897,370.901,-146.565,172.163,49.096,159.783
C08812=1022.888,370.655,-146.525,172.154,49.096,159.782
C08813=1022.880,370.408,-146.485,172.146,49.096,159.780
C08814=1022.871,370.161,-146.445,172.138,49.096,159.779
C08815=1022.863,369.914,-146.405,172.129,49.096,159.778
C08816=1022.855,369.668,-146.366,172.121,49.096,159.777
C08817=1022.847,369.422,-146.325,172.113,49.096,159.776
C08818=1022.838,369.175,-146.286,172.104,49.096,159.774
C08819=1022.831,368.928,-146.246,172.096,49.096,159.773
C08820=1022.822,368.681,-146.206,172.088,49.096,159.772
C08821=1022.814,368.434,-146.165,172.079,49.096,159.770
C08822=1022.805,368.188,-146.126,172.071,49.097,159.769
C08823=1022.797,367.941,-146.087,172.063,49.097,159.768
C08824=1022.789,367.694,-146.047,172.055,49.097,159.767
C08825=1022.780,367.454,-146.009,172.047,49.097,159.766
C08826=1022.772,367.214,-145.970,172.038,49.097,159.764
C08827=1022.765,366.973,-145.932,172.031,49.097,159.763
C08828=1022.756,366.734,-145.893,172.023,49.098,159.762
C08829=1022.748,366.493,-145.855,172.015,49.098,159.761
C08830=1022.740,366.253,-145.817,172.007,49.099,159.760
C08831=1022.732,366.013,-145.779,171.999,49.098,159.759
C08832=1022.724,365.772,-145.741,171.991,49.099,159.757
C08833=1022.716,365.526,-145.701,171.983,49.099,159.756
C08834=1022.708,365.279,-145.663,171.975,49.099,159.755
C08835=1022.700,365.032,-145.623,171.967,49.100,159.754
C08836=1022.691,364.785,-145.583,171.959,49.100,159.753
C08837=1022.683,364.539,-145.544,171.951,49.100,159.752
C08838=1022.675,364.291,-145.505,171.943,49.100,159.750
C08839=1022.666,364.045,-145.466,171.935,49.101,159.749
C08840=1022.658,363.798,-145.428,171.927,49.101,159.748
C08841=1022.651,363.551,-145.388,171.919,49.101,159.747
C08842=1022.643,363.305,-145.349,171.911,49.102,159.746
C08843=1022.634,363.058,-145.310,171.904,49.102,159.745
C08844=1022.626,362.811,-145.271,171.896,49.102,159.744
C08845=1022.618,362.564,-145.232,171.888,49.103,159.743
C08846=1022.610,362.317,-145.194,171.880,49.103,159.741
C08847=1022.603,362.070,-145.154,171.872,49.104,159.741
C08848=1022.594,361.823,-145.115,171.865,49.104,159.739
C08849=1022.586,361.576,-145.076,171.857,49.105,159.738
C08850=1022.578,361.330,-145.038,171.849,49.105,159.737
C08851=1022.570,361.083,-144.999,171.841,49.106,159.736
C08852=1022.562,360.836,-144.960,171.833,49.106,159.735
C08853=1022.555,360.589,-144.921,171.826,49.107,159.734
C08854=1022.547,360.342,-144.882,171.818,49.107,159.733
C08855=1022.539,360.095,-144.844,171.810,49.107,159.732
C08856=1022.531,359.849,-144.805,171.802,49.108,159.731
C08857=1022.523,359.602,-144.766,171.795,49.109,159.730
C08858=1022.515,359.355,-144.728,171.787,49.109,159.729
C08859=1022.507,359.108,-144.689,171.780,49.110,159.728
C08860=1022.499,358.861,-144.651,171.772,49.110,159.727
C08861=1022.491,358.614,-144.613,171.764,49.111,159.726
C08862=1022.482,358.367,-144.575,171.757,49.111,159.725
C08863=1022.475,358.121,-144.536,171.749,49.112,159.724
C08864=1022.467,357.873,-144.498,171.741,49.113,159.723
C08865=1022.459,357.627,-144.460,171.734,49.114,159.722
C08866=1022.451,357.379,-144.422,171.726,49.114,159.721
C08867=1022.443,357.132,-144.383,171.719,49.115,159.720
C08868=1022.436,356.886,-144.345,171.711,49.115,159.719
C08869=1022.428,356.638,-144.307,171.704,49.116,159.718
C08870=1022.419,356.392,-144.269,171.696,49.117,159.717
C08871=1022.412,356.145,-144.231,171.689,49.117,159.716
C08872=1022.404,355.898,-144.192,171.681,49.118,159.715
C08873=1022.396,355.651,-144.155,171.673,49.119,159.714
C08874=1022.388,355.404,-144.116,171.667,49.120,159.713
C08875=1022.381,355.156,-144.079,171.659,49.120,159.712
C08876=1022.373,354.910,-144.041,171.652,49.121,159.711
C08877=1022.365,354.663,-144.002,171.644,49.122,159.710
C08878=1022.357,354.416,-143.965,171.636,49.123,159.709
C08879=1022.349,354.169,-143.926,171.630,49.124,159.708
C08880=1022.341,353.922,-143.889,171.622,49.125,159.707
C08881=1022.334,353.675,-143.852,171.615,49.126,159.706
C08882=1022.326,353.427,-143.813,171.607,49.126,159.705
C08883=1022.318,353.181,-143.776,171.599,49.127,159.704
C08884=1022.311,352.933,-143.739,171.593,49.128,159.703
C08885=1022.303,352.696,-143.702,171.585,49.129,159.703
C08886=1022.295,352.460,-143.667,171.578,49.130,159.702
C08887=1022.288,352.223,-143.630,171.572,49.131,159.701
C08888=1022.281,351.986,-143.594,171.565,49.131,159.700
C08889=1022.274,351.750,-143.558,171.557,49.132,159.699
C08890=1022.265,351.512,-143.522,171.550,49.133,159.698
C08891=1022.258,351.275,-143.486,171.544,49.134,159.697
C08892=1022.251,351.039,-143.450,171.537,49.135,159.697
C08893=1022.243,350.792,-143.413,171.530,49.136,159.696
C08894=1022.236,350.545,-143.376,171.523,49.137,159.695
C08895=1022.228,350.297,-143.338,171.515,49.138,159.694
C08896=1022.220,350.050,-143.301,171.508,49.139,159.693
C08897=1022.213,349.803,-143.263,171.501,49.140,159.692
C08898=1022.206,349.556,-143.226,171.494,49.141,159.691
C08899=1022.198,349.309,-143.189,171.487,49.142,159.691
C08900=1022.190,349.062,-143.151,171.480,49.143,159.690
C08901=1022.183,348.815,-143.114,171.472,49.144,159.689
C08902=1022.175,348.568,-143.077,171.466,49.145,159.688
C08903=1022.168,348.321,-143.039,171.458,49.147,159.687
C08904=1022.160,348.074,-143.002,171.452,49.147,159.686
C08905=1022.153,347.827,-142.965,171.444,49.148,159.686
C08906=1022.145,347.579,-142.929,171.437,49.150,159.685
C08907=1022.138,347.332,-142.891,171.430,49.151,159.684
C08908=1022.130,347.086,-142.854,171.423,49.152,159.683
C08909=1022.123,346.838,-142.817,171.416,49.153,159.682
C08910=1022.115,346.591,-142.780,171.409,49.154,159.682
C08911=1022.107,346.344,-142.743,171.402,49.155,159.681
C08912=1022.100,346.096,-142.707,171.395,49.157,159.680
C08913=1022.092,345.850,-142.670,171.389,49.158,159.679
C08914=1022.084,345.602,-142.633,171.381,49.159,159.678
C08915=1022.077,345.355,-142.596,171.375,49.160,159.678
C08916=1022.069,345.108,-142.560,171.367,49.162,159.677
C08917=1022.062,344.860,-142.522,171.360,49.163,159.676
C08918=1022.054,344.613,-142.486,171.354,49.164,159.675
C08919=1022.046,344.366,-142.449,171.347,49.166,159.675
C08920=1022.040,344.118,-142.412,171.340,49.166,159.674
C08921=1022.032,343.872,-142.375,171.333,49.168,159.673
C08922=1022.024,343.625,-142.339,171.326,49.169,159.672
C08923=1022.018,343.377,-142.303,171.320,49.171,159.672
C08924=1022.010,343.130,-142.266,171.312,49.172,159.671
C08925=1022.002,342.883,-142.229,171.306,49.173,159.670
C08926=1021.995,342.635,-142.193,171.299,49.174,159.670
C08927=1021.987,342.388,-142.156,171.292,49.176,159.669
C08928=1021.980,342.141,-142.120,171.285,49.177,159.668
C08929=1021.973,341.894,-142.083,171.279,49.178,159.667
C08930=1021.965,341.646,-142.047,171.272,49.180,159.667
C08931=1021.958,341.399,-142.011,171.265,49.181,159.666
C08932=1021.950,341.153,-141.974,171.259,49.183,159.665
C08933=1021.943,340.905,-141.937,171.252,49.184,159.665
C08934=1021.936,340.657,-141.901,171.245,49.186,159.664
C08935=1021.929,340.411,-141.865,171.239,49.187,159.663
C08936=1021.921,340.163,-141.829,171.231,49.189,159.663
C08937=1021.914,339.916,-141.792,171.225,49.190,159.662
C08938=1021.907,339.669,-141.756,171.219,49.191,159.661
C08939=1021.899,339.421,-141.720,171.211,49.193,159.660
C08940=1021.891,339.174,-141.684,171.205,49.194,159.660
C08941=1021.884,338.927,-141.648,171.198,49.196,159.659
C08942=1021.877,338.679,-141.613,171.191,49.197,159.658
C08943=1021.869,338.432,-141.576,171.185,49.199,159.658
C08944=1021.862,338.185,-141.540,171.179,49.200,159.657
